# B&R Automation Studio project ACOPOStrak
Automation Studio 4.7.4.67 SP; technology packages: mapp 5.9.1, mappCockpit 5.9.0, mappMotion 5.9.2, mappView 5.9.1

## Configuration ACOPOStrak

### IoMap.iom - 5PC900_TS17_00/IoMap.iom
```iecst
VAR_CONFIG
	::gMain.status.safety.moduleOK AT %IX."epl_icn".ModuleOk;
	::gMain.status.safety.resetNeeded AT %IX."epl_icn".resetNeeded;
	::gMain.cmd.safety.reset AT %QX."epl_icn".resetCommand;
	::gMain.status.safety.started AT %IX."epl_icn".safetyStarted;
	::gMain.status.safety.ready AT %IX."epl_icn".safetyOK;
END_VAR
```

## Configuration Safety

CPU X20CP0484, AutomationRuntime C4.72, Build 4.1.2, Safety 0.0, Vc V4.72.0

### Task classes (Cpu.sw)
```
Cyclic#2 (cycle 20000 us, tolerance 20000 us):
  Safety <- Modules.Safety.Safety.prg
Binaries: arsvcreg, udbdef, TCData, arflatprv, arcoal, mvLoader, FWRules, mCoWebSc, ashwd, ashwac, User, sysconf, asfw, arconfig, Role, iomap, Config
Libraries: DataObj, AsXml, standard, runtime, FileIO, astime, mpbase, SfDomVis, asiodiag, asieccon, aruser, brsystem, SfDomDrv, sys_lib, MpSfDomMgr, asusb, astcp
```

### Hardware
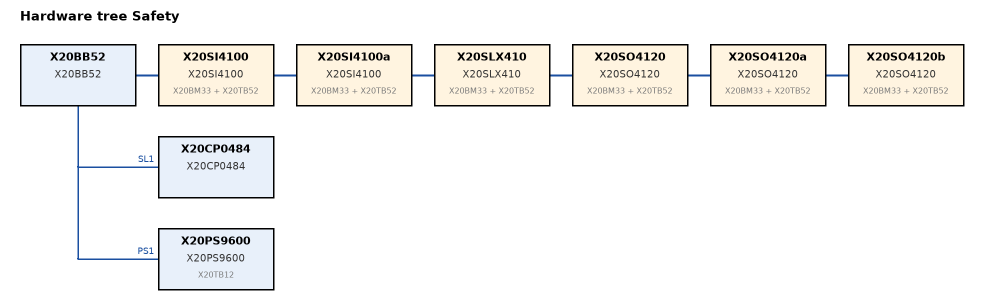
```
X20BB52 : X20BB52 v1.1.0.0
X20BM33 : X20BM33 v1.0.0.6  [X2X1 -> X20BB52.IF6]
X20BM33a : X20BM33 v1.0.0.6  [X2X1 -> X20BM33.X2X2]
X20BM33b : X20BM33 v1.0.0.6  [X2X1 -> X20BM33a.X2X2]
X20BM33c : X20BM33 v1.0.0.6  [X2X1 -> X20BM33b.X2X2]
X20BM33d : X20BM33 v1.0.0.6  [X2X1 -> X20BM33c.X2X2]
X20BM33e : X20BM33 v1.0.0.6  [X2X1 -> X20BM33d.X2X2]
X20CP0484 : X20CP0484 v1.2.1.0  [SL -> X20BB52.SL1]
  Connector IF2:
    ActivateDevice = 1
    Mode = Manual
    InternetAddress = 192.168.1.200
    SubnetMask = 255.255.255.0
  Connector IF3:
    CycleTime = 2400
    Mode = CN
    NodeID = 200
    EplNatSubnet = 192.168.103.0
    Channel1
    ChannelID1 = safetyStarted
    ChannelDirection1 = OUT
    Channel2
    ChannelID2 = safetyOK
    ChannelDirection2 = OUT
    Channel3
    ChannelID3 = resetNeeded
    ChannelDirection3 = OUT
    Channel4
    ChannelID4 = resetCommand
  ConfigurationID = ACOPOStrak_Safety
  TimerDeviceType = SWIOTIMER
  Cyclic1Duration = 2400
  Cyclic1Tolerance = 0
  Cyclic2Duration = 20000
  Cyclic2Tolerance = 20000
  Cyclic3Duration = 50000
  Cyclic3Tolerance = 50000
  Cyclic4Duration = 100000
  Cyclic4Tolerance = 100000
  Cyclic5Duration = 200000
  Cyclic5Tolerance = 200000
  Cyclic6Duration = 500000
  Cyclic6Tolerance = 500000
  Cyclic7Duration = 1000000
  Cyclic7Tolerance = 1000000
  Cyclic8Duration = 10000
  Cyclic8Tolerance = 30000000
X20PS9600 : X20PS9600 v1.0.1.0  [PS -> X20BB52.PS1; SS1 -> X20TB12.SS]
X20SI4100 : X20SI4100 v1.10.9.1  [SS1 -> X20TB52.SS; SL -> X20BM33.SL1]
  Supervision = off
X20SI4100a : X20SI4100 v1.10.9.1  [SS1 -> X20TB52a.SS; SL -> X20BM33a.SL1]
  Supervision = off
  SafeModuleID = 3
X20SLX410 : X20SLX410 v1.10.10.4  [SS1 -> X20TB52b.SS; SL -> X20BM33b.SL1]
  Supervision = off
X20SO4120 : X20SO4120 v1.10.9.1  [SS1 -> X20TB52c.SS; SL -> X20BM33c.SL1]
  Supervision = off
  SafeModuleID = 4
  DigitalOutput01 = viaSafeLOGIC
  DigitalOutput02 = viaSafeLOGIC
  DigitalOutput03 = viaSafeLOGIC
  DigitalOutput04 = viaSafeLOGIC
X20SO4120a : X20SO4120 v1.10.9.1  [SS1 -> X20TB52d.SS; SL -> X20BM33d.SL1]
  Supervision = off
  SafeModuleID = 5
  DigitalOutput01 = viaSafeLOGIC
  DigitalOutput02 = viaSafeLOGIC
  DigitalOutput03 = viaSafeLOGIC
  DigitalOutput04 = viaSafeLOGIC
X20SO4120b : X20SO4120 v1.10.9.1  [SS1 -> X20TB52e.SS; SL -> X20BM33e.SL1]
  Supervision = off
  SafeModuleID = 6
  DigitalOutput01 = viaSafeLOGIC
  DigitalOutput02 = viaSafeLOGIC
  DigitalOutput03 = viaSafeLOGIC
  DigitalOutput04 = viaSafeLOGIC
X20TB12 : X20TB12 v1.0.0.0
X20TB52 : X20TB52 v1.0.0.1
X20TB52a : X20TB52 v1.0.0.1
X20TB52b : X20TB52 v1.0.0.1
X20TB52c : X20TB52 v1.0.0.1
X20TB52d : X20TB52 v1.0.0.1
X20TB52e : X20TB52 v1.0.0.1
```

### IoMap.iom - X20CP0484/IoMap.iom
```iecst
VAR_CONFIG
	::Safety:this.cmd.reset AT %QX."X20SLX410".BOOL10001;
	::Safety:this.status.safetyStarted AT %IX."X20SLX410".BOOL00001;
	::Safety:this.status.safetyOk AT %IX."X20SLX410".BOOL00002;
	::Safety:this.status.resetNeeded AT %IX."X20SLX410".BOOL00003;
	::Safety:this.status.safetyStarted AT %QX."X20CP0484".IF3.safetyStarted;
	::Safety:this.status.safetyOk AT %QX."X20CP0484".IF3.safetyOK;
	::Safety:this.status.resetNeeded AT %QX."X20CP0484".IF3.resetNeeded;
	::Safety:this.cmd.reset AT %IX."X20CP0484".IF3.resetCommand;
END_VAR
```

- Safety project (password-protected, skipped)

## Configuration Simulation

CPU 5PC900.TS17-00, AutomationRuntime C4.72, Build 4.1.2, Safety 0.0, Vc V4.53.0

### Task classes (Cpu.sw)
```
Cyclic#1:
  Main <- Modules.Main.Main.prg
  Track1Sect <- Modules.Sectors.Track1Sector.Track1Sector.prg  // Task for handling Track 1 sectors
  Track2Sect <- Modules.Sectors.Track2Sector.Track2Sector.prg
  Track3Sect <- Modules.Sectors.Track3Sector.Track3Sector.prg  // Task for handling Track 3 sectors
  Track4Sect <- Modules.Sectors.Track4Sector.Track4Sector.prg  // Task for handling Track 4 sectors
  Track5Sect <- Modules.Sectors.Track5Sector.Track5Sector.prg
  Track6Sect <- Modules.Sectors.Track6Sector.Track6Sector.prg
Cyclic#8:
  Alarm <- Services.Alarm.Alarm.prg
  Simulation <- Simulation.Simulation.prg
DataObjects: McAcpSys
Binaries: TCData, udbdef, mvLoader, mCoWebSc, McAcpSim, arsvcreg, McAcpDrv, McProfGen, arflatprv, arcoal, Config_5, Config_4, AlarmCore, AlarmHist, Settings, ashwac, arconfig, asfw, TraceConfi, User, ashwd, iomap, Role, sysconf, Config_1, Config_3, Config_2
Libraries: McAxis, McBase, McAcpTrak, brdkMU, brsystem, AsSem, sys_lib, runtime, brdkSTR, operator, astime, AsIecCon, CoTrace, AsZip, FileIO, MpAlarmX, MpBase, MpAxis, McAcpAx, AsBrStr, AsIODiag, powerlnk, dataobj, MpSfDomMgr, SfDomDrv, SfDomVis, aruser, asusb, standard, astcp
```

### Hardware
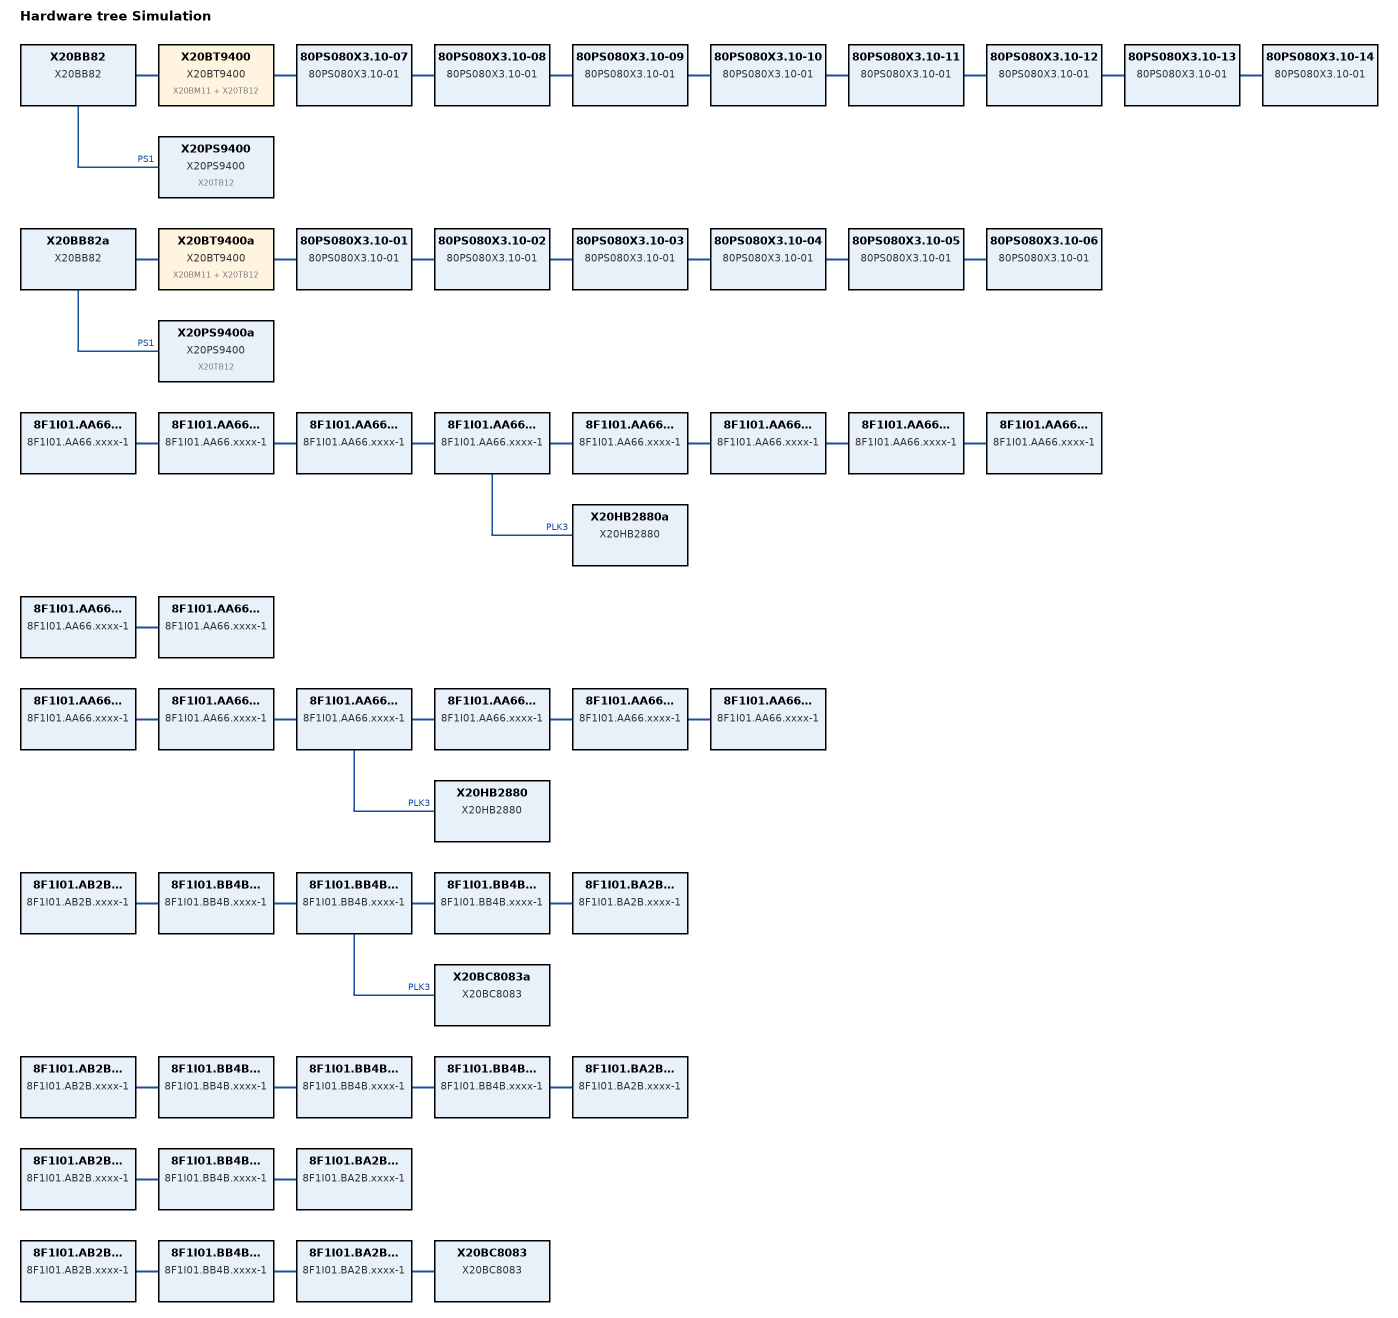
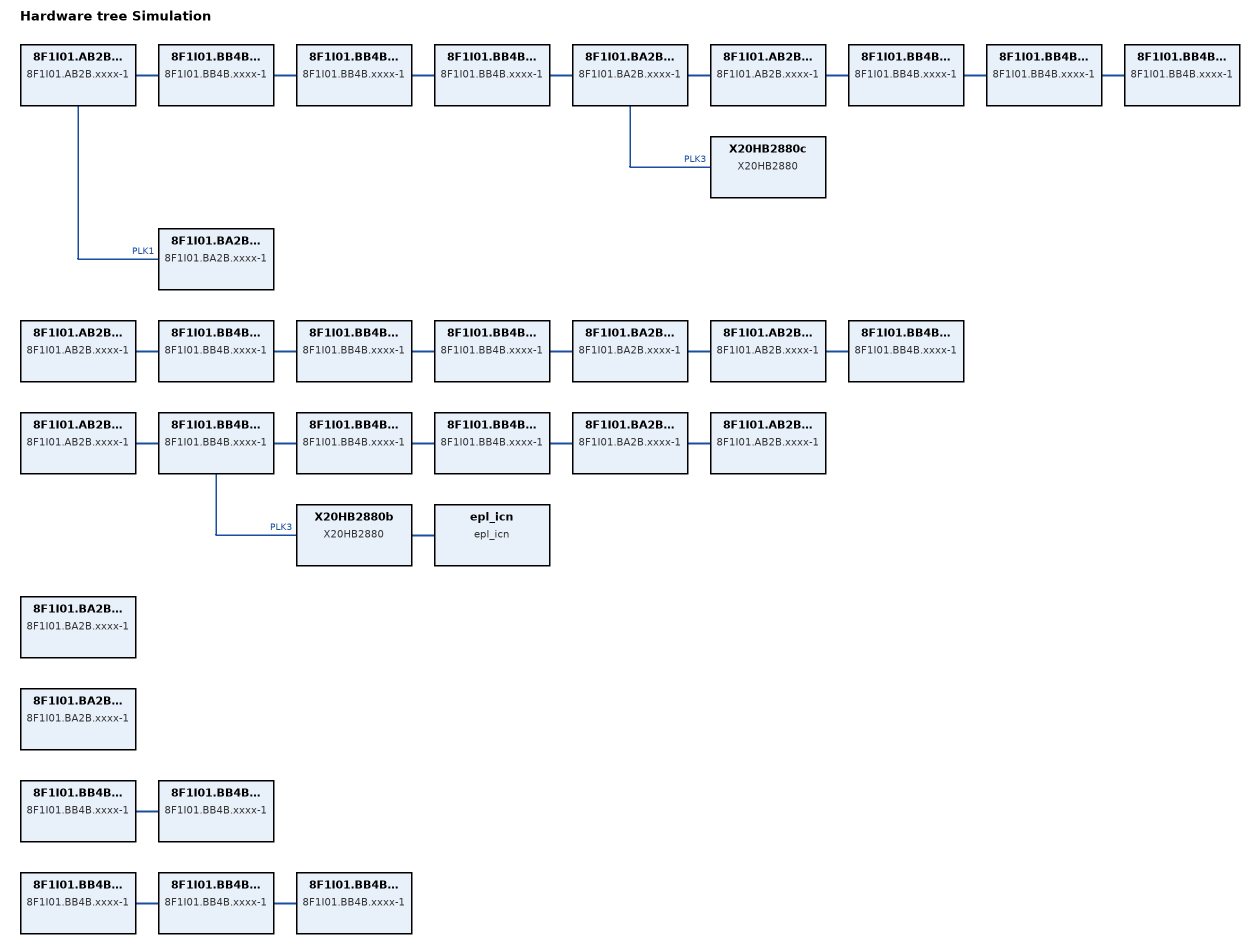
```
80PS080X3.10-01 : 80PS080X3.10-01 v1.3.0.0  [X2X1 -> X20BT9400a.X2X1 [Cable Type=X2XCable, Length=3, Version=1.0.0.2]]
  Supervision = off
  ParallelMode01 = on
  VoltageSet01 = 60
  ChopperEnable01 = on
80PS080X3.10-02 : 80PS080X3.10-01 v1.3.0.0  [X2X1 -> 80PS080X3.10-01.X2X2 [Cable Type=X2XCable, Length=1, Version=1.0.0.2]]
  Supervision = off
  ParallelMode01 = on
  VoltageSet01 = 60
  ChopperEnable01 = on
80PS080X3.10-03 : 80PS080X3.10-01 v1.3.0.0  [X2X1 -> 80PS080X3.10-02.X2X2 [Cable Type=X2XCable, Length=5, Version=1.0.0.2]]
  Supervision = off
  VoltageSet01 = 58
  ChopperEnable01 = on
80PS080X3.10-04 : 80PS080X3.10-01 v1.3.0.0  [X2X1 -> 80PS080X3.10-03.X2X2 [Cable Type=X2XCable, Length=1, Version=1.0.0.2]]
  Supervision = off
  VoltageSet01 = 58
  ChopperEnable01 = on
80PS080X3.10-05 : 80PS080X3.10-01 v1.3.0.0  [X2X1 -> 80PS080X3.10-04.X2X2 [Cable Type=X2XCable, Length=5, Version=1.0.0.2]]
  Supervision = off
  VoltageSet01 = 58
  ChopperEnable01 = on
80PS080X3.10-06 : 80PS080X3.10-01 v1.3.0.0  [X2X1 -> 80PS080X3.10-05.X2X2 [Cable Type=X2XCable, Length=1, Version=1.0.0.2]]
  Supervision = off
  VoltageSet01 = 58
  ChopperEnable01 = on
80PS080X3.10-07 : 80PS080X3.10-01 v1.3.0.0  [X2X1 -> X20BT9400.X2X1 [Cable Type=X2XCable, Length=5, Version=1.0.0.2]]
  Supervision = off
  VoltageSet01 = 58
  ChopperEnable01 = on
80PS080X3.10-08 : 80PS080X3.10-01 v1.3.0.0  [X2X1 -> 80PS080X3.10-07.X2X2 [Cable Type=X2XCable, Length=1, Version=1.0.0.2]]
  Supervision = off
  VoltageSet01 = 58
  ChopperEnable01 = on
80PS080X3.10-09 : 80PS080X3.10-01 v1.3.0.0  [X2X1 -> 80PS080X3.10-08.X2X2 [Cable Type=X2XCable, Length=1, Version=1.0.0.2]]
  Supervision = off
  VoltageSet01 = 58
  ChopperEnable01 = on
80PS080X3.10-10 : 80PS080X3.10-01 v1.3.0.0  [X2X1 -> 80PS080X3.10-09.X2X2 [Cable Type=X2XCable, Length=1, Version=1.0.0.2]]
  Supervision = off
  VoltageSet01 = 58
  ChopperEnable01 = on
80PS080X3.10-11 : 80PS080X3.10-01 v1.3.0.0  [X2X1 -> 80PS080X3.10-10.X2X2 [Cable Type=X2XCable, Length=3, Version=1.0.0.2]]
  Supervision = off
  VoltageSet01 = 58
  ChopperEnable01 = on
80PS080X3.10-12 : 80PS080X3.10-01 v1.3.0.0  [X2X1 -> 80PS080X3.10-11.X2X2 [Cable Type=X2XCable, Length=1, Version=1.0.0.2]]
  Supervision = off
  VoltageSet01 = 58
  ChopperEnable01 = on
80PS080X3.10-13 : 80PS080X3.10-01 v1.3.0.0  [X2X1 -> 80PS080X3.10-12.X2X2 [Cable Type=X2XCable, Length=1, Version=1.0.0.2]]
  Supervision = off
  VoltageSet01 = 58
  ChopperEnable01 = on
80PS080X3.10-14 : 80PS080X3.10-01 v1.3.0.0  [X2X1 -> 80PS080X3.10-13.X2X2 [Cable Type=X2XCable, Length=1, Version=1.0.0.2]]
  Supervision = off
  VoltageSet01 = 58
  ChopperEnable01 = on
8F1I01.AA66.xxxx-16 : 8F1I01.AA66.xxxx-1 v1.0.0.1  [PLK2 -> 8F1I01.AA66.xxxx-17.PLK1 (NodeNumber=16) [Cable Type=PowerlinkCable, Length=10, Version=1.0.0.2]]
  DriveConfiguration:
    McTypeID = LLMConfig
  DriveConfiguration/Segment:
    Shape = STRAIGHT660
    SegmentReference = SEG_1_16
    StopReaction = UseAssemblySetting
    SpeedFilter = UseAssemblySetting
8F1I01.AA66.xxxx-17 : 8F1I01.AA66.xxxx-1 v1.0.0.1  [PLK1 -> 8F1I01.AA66.xxxx-16.PLK2 (NodeNumber=17) [Cable Type=PowerlinkCable, Length=10, Version=1.0.0.2]; PLK2 -> 8F1I01.AA66.xxxx-18.PLK1 (NodeNumber=17) [Cable Type=PowerlinkCable, Length=10, Version=1.0.0.2]]
  DriveConfiguration:
    McTypeID = LLMConfig
  DriveConfiguration/Segment:
    Shape = STRAIGHT660
    SegmentReference = SEG_1_17
    StopReaction = UseAssemblySetting
    SpeedFilter = UseAssemblySetting
8F1I01.AA66.xxxx-18 : 8F1I01.AA66.xxxx-1 v1.0.0.1  [PLK1 -> 8F1I01.AA66.xxxx-17.PLK2 (NodeNumber=18) [Cable Type=PowerlinkCable, Length=10, Version=1.0.0.2]; PLK2 -> 8F1I01.AA66.xxxx-19.PLK1 (NodeNumber=18) [Cable Type=PowerlinkCable, Length=10, Version=1.0.0.2]]
  DriveConfiguration:
    McTypeID = LLMConfig
  DriveConfiguration/Segment:
    Shape = STRAIGHT660
    SegmentReference = SEG_1_18
    StopReaction = UseAssemblySetting
    SpeedFilter = UseAssemblySetting
8F1I01.AA66.xxxx-19 : 8F1I01.AA66.xxxx-1 v1.0.0.1  [PLK1 -> 8F1I01.AA66.xxxx-18.PLK2 (NodeNumber=19) [Cable Type=PowerlinkCable, Length=10, Version=1.0.0.2]; PLK2 -> 8F1I01.AA66.xxxx-20.PLK1 (NodeNumber=19) [Cable Type=PowerlinkCable, Length=10, Version=1.0.0.2]; PLK3 -> X20HB2880a.ETH1 (NodeNumber=19) [Cable Type=PowerlinkCable, Length=10, Version=1.0.0.2]]
  DriveConfiguration:
    McTypeID = LLMConfig
  DriveConfiguration/Segment:
    Shape = STRAIGHT660
    SegmentReference = SEG_1_19
    StopReaction = UseAssemblySetting
    SpeedFilter = UseAssemblySetting
8F1I01.AA66.xxxx-20 : 8F1I01.AA66.xxxx-1 v1.0.0.1  [PLK1 -> 8F1I01.AA66.xxxx-19.PLK2 (NodeNumber=20) [Cable Type=PowerlinkCable, Length=10, Version=1.0.0.2]; PLK2 -> 8F1I01.AA66.xxxx-21.PLK1 (NodeNumber=20) [Cable Type=PowerlinkCable, Length=10, Version=1.0.0.2]]
  DriveConfiguration:
    McTypeID = LLMConfig
  DriveConfiguration/Segment:
    Shape = STRAIGHT660
    SegmentReference = SEG_1_20
    StopReaction = UseAssemblySetting
    SpeedFilter = UseAssemblySetting
8F1I01.AA66.xxxx-21 : 8F1I01.AA66.xxxx-1 v1.0.0.1  [PLK1 -> 8F1I01.AA66.xxxx-20.PLK2 (NodeNumber=21) [Cable Type=PowerlinkCable, Length=10, Version=1.0.0.2]; PLK2 -> 8F1I01.AA66.xxxx-22.PLK1 (NodeNumber=21) [Cable Type=PowerlinkCable, Length=10, Version=1.0.0.2]]
  DriveConfiguration:
    McTypeID = LLMConfig
  DriveConfiguration/Segment:
    Shape = STRAIGHT660
    SegmentReference = SEG_1_21
    StopReaction = UseAssemblySetting
    SpeedFilter = UseAssemblySetting
8F1I01.AA66.xxxx-22 : 8F1I01.AA66.xxxx-1 v1.0.0.1  [PLK1 -> 8F1I01.AA66.xxxx-21.PLK2 (NodeNumber=22) [Cable Type=PowerlinkCable, Length=10, Version=1.0.0.2]; PLK2 -> 8F1I01.AA66.xxxx-23.PLK1 (NodeNumber=22) [Cable Type=PowerlinkCable, Length=10, Version=1.0.0.2]]
  DriveConfiguration:
    McTypeID = LLMConfig
  DriveConfiguration/Segment:
    Shape = STRAIGHT660
    SegmentReference = SEG_1_22
    StopReaction = UseAssemblySetting
    SpeedFilter = UseAssemblySetting
8F1I01.AA66.xxxx-23 : 8F1I01.AA66.xxxx-1 v1.0.0.1  [PLK1 -> 8F1I01.AA66.xxxx-22.PLK2 (NodeNumber=23) [Cable Type=PowerlinkCable, Length=10, Version=1.0.0.2]]
  DriveConfiguration:
    McTypeID = LLMConfig
  DriveConfiguration/Segment:
    Shape = STRAIGHT660
    SegmentReference = SEG_1_23
    StopReaction = UseAssemblySetting
    SpeedFilter = UseAssemblySetting
8F1I01.AA66.xxxx-29 : 8F1I01.AA66.xxxx-1 v1.0.0.1  [PLK1 -> 8F1I01.BA2B.xxxx-28.PLK2 (NodeNumber=29) [Cable Type=PowerlinkCable, Length=10, Version=1.0.0.2]; PLK2 -> 8F1I01.AA66.xxxx-30.PLK1 (NodeNumber=29) [Cable Type=PowerlinkCable, Length=10, Version=1.0.0.2]]
  DriveConfiguration:
    McTypeID = LLMConfig
  DriveConfiguration/Segment:
    Shape = STRAIGHT660
    SegmentReference = SEG_1_29
    StopReaction = UseAssemblySetting
    SpeedFilter = UseAssemblySetting
8F1I01.AA66.xxxx-30 : 8F1I01.AA66.xxxx-1 v1.0.0.1  [PLK1 -> 8F1I01.AA66.xxxx-29.PLK2 (NodeNumber=30) [Cable Type=PowerlinkCable, Length=10, Version=1.0.0.2]]
  DriveConfiguration:
    McTypeID = LLMConfig
  DriveConfiguration/Segment:
    Shape = STRAIGHT660
    SegmentReference = SEG_1_30
    StopReaction = UseAssemblySetting
    SpeedFilter = UseAssemblySetting
8F1I01.AA66.xxxx-31 : 8F1I01.AA66.xxxx-1 v1.0.0.1  [PLK2 -> 8F1I01.AA66.xxxx-32.PLK1 (NodeNumber=31) [Cable Type=PowerlinkCable, Length=10, Version=1.0.0.2]]
  DriveConfiguration:
    McTypeID = LLMConfig
  DriveConfiguration/Segment:
    Shape = STRAIGHT660
    SegmentReference = SEG_1_31
    StopReaction = UseAssemblySetting
    SpeedFilter = UseAssemblySetting
8F1I01.AA66.xxxx-32 : 8F1I01.AA66.xxxx-1 v1.0.0.1  [PLK1 -> 8F1I01.AA66.xxxx-31.PLK2 (NodeNumber=32) [Cable Type=PowerlinkCable, Length=10, Version=1.0.0.2]; PLK2 -> 8F1I01.AA66.xxxx-33.PLK1 (NodeNumber=32) [Cable Type=PowerlinkCable, Length=10, Version=1.0.0.2]]
  DriveConfiguration:
    McTypeID = LLMConfig
  DriveConfiguration/Segment:
    Shape = STRAIGHT660
    SegmentReference = SEG_1_32
    StopReaction = UseAssemblySetting
    SpeedFilter = UseAssemblySetting
8F1I01.AA66.xxxx-33 : 8F1I01.AA66.xxxx-1 v1.0.0.1  [PLK1 -> 8F1I01.AA66.xxxx-32.PLK2 (NodeNumber=33) [Cable Type=PowerlinkCable, Length=10, Version=1.0.0.2]; PLK2 -> 8F1I01.AA66.xxxx-34.PLK1 (NodeNumber=33) [Cable Type=PowerlinkCable, Length=10, Version=1.0.0.2]; PLK3 -> X20HB2880.ETH1 (NodeNumber=33) [Cable Type=PowerlinkCable, Length=10, Version=1.0.0.2]]
  DriveConfiguration:
    McTypeID = LLMConfig
  DriveConfiguration/Segment:
    Shape = STRAIGHT660
    SegmentReference = SEG_1_33
    StopReaction = UseAssemblySetting
    SpeedFilter = UseAssemblySetting
8F1I01.AA66.xxxx-34 : 8F1I01.AA66.xxxx-1 v1.0.0.1  [PLK1 -> 8F1I01.AA66.xxxx-33.PLK2 (NodeNumber=34) [Cable Type=PowerlinkCable, Length=10, Version=1.0.0.2]; PLK2 -> 8F1I01.AA66.xxxx-35.PLK1 (NodeNumber=34) [Cable Type=PowerlinkCable, Length=10, Version=1.0.0.2]]
  DriveConfiguration:
    McTypeID = LLMConfig
  DriveConfiguration/Segment:
    Shape = STRAIGHT660
    SegmentReference = SEG_1_34
    StopReaction = UseAssemblySetting
    SpeedFilter = UseAssemblySetting
8F1I01.AA66.xxxx-35 : 8F1I01.AA66.xxxx-1 v1.0.0.1  [PLK1 -> 8F1I01.AA66.xxxx-34.PLK2 (NodeNumber=35) [Cable Type=PowerlinkCable, Length=10, Version=1.0.0.2]; PLK2 -> 8F1I01.AA66.xxxx-36.PLK1 (NodeNumber=35) [Cable Type=PowerlinkCable, Length=10, Version=1.0.0.2]]
  DriveConfiguration:
    McTypeID = LLMConfig
  DriveConfiguration/Segment:
    Shape = STRAIGHT660
    SegmentReference = SEG_1_35
    StopReaction = UseAssemblySetting
    SpeedFilter = UseAssemblySetting
8F1I01.AA66.xxxx-36 : 8F1I01.AA66.xxxx-1 v1.0.0.1  [PLK1 -> 8F1I01.AA66.xxxx-35.PLK2 (NodeNumber=36) [Cable Type=PowerlinkCable, Length=10, Version=1.0.0.2]]
  DriveConfiguration:
    McTypeID = LLMConfig
  DriveConfiguration/Segment:
    Shape = STRAIGHT660
    SegmentReference = SEG_1_36
    StopReaction = UseAssemblySetting
    SpeedFilter = UseAssemblySetting
8F1I01.AB2B.xxxx-11 : 8F1I01.AB2B.xxxx-1 v1.0.0.1  [PLK2 -> 8F1I01.BB4B.xxxx-12.PLK1 (NodeNumber=11) [Cable Type=PowerlinkCable, Length=10, Version=1.0.0.2]]
  DriveConfiguration:
    McTypeID = LLMConfig
  DriveConfiguration/Segment:
    Shape = STRAIGHT105_TO_CIRCULAR
    SegmentReference = SEG_1_11
    StopReaction = UseAssemblySetting
    SpeedFilter = UseAssemblySetting
8F1I01.AB2B.xxxx-24 : 8F1I01.AB2B.xxxx-1 v1.0.0.1  [PLK2 -> 8F1I01.BB4B.xxxx-25.PLK1 (NodeNumber=24) [Cable Type=PowerlinkCable, Length=10, Version=1.0.0.2]]
  DriveConfiguration:
    McTypeID = LLMConfig
  DriveConfiguration/Segment:
    Shape = STRAIGHT105_TO_CIRCULAR
    SegmentReference = SEG_1_24
    StopReaction = UseAssemblySetting
    SpeedFilter = UseAssemblySetting
8F1I01.AB2B.xxxx-37 : 8F1I01.AB2B.xxxx-1 v1.0.0.1  [PLK2 -> 8F1I01.BB4B.xxxx-38.PLK1 (NodeNumber=37) [Cable Type=PowerlinkCable, Length=10, Version=1.0.0.2]; PLK3 -> X20HB2880.ETH2 (NodeNumber=37) [Cable Type=PowerlinkCable, Length=10, Version=1.0.0.2]]
  DriveConfiguration:
    McTypeID = LLMConfig
  DriveConfiguration/Segment:
    Shape = STRAIGHT105_TO_CIRCULAR
    SegmentReference = SEG_5_37
    StopReaction = UseAssemblySetting
    SpeedFilter = UseAssemblySetting
8F1I01.AB2B.xxxx-51 : 8F1I01.AB2B.xxxx-1 v1.0.0.1  [PLK2 -> 8F1I01.BB4B.xxxx-52.PLK1 (NodeNumber=51) [Cable Type=PowerlinkCable, Length=10, Version=1.0.0.2]]
  DriveConfiguration:
    McTypeID = LLMConfig
  DriveConfiguration/Segment:
    Shape = STRAIGHT105_TO_CIRCULAR
    SegmentReference = SEG_6_51
    StopReaction = UseAssemblySetting
    SpeedFilter = UseAssemblySetting
8F1I01.AB2B.xxxx-55 : 8F1I01.AB2B.xxxx-1 v1.0.0.1  [PLK1 -> 8F1I01.BA2B.xxxx-54.PLK2 (NodeNumber=55) [Cable Type=PowerlinkCable, Length=10, Version=1.0.0.2]; PLK2 -> 8F1I01.BB4B.xxxx-56.PLK1 (NodeNumber=55) [Cable Type=PowerlinkCable, Length=10, Version=1.0.0.2]]
  DriveConfiguration:
    McTypeID = LLMConfig
  DriveConfiguration/Segment:
    Shape = STRAIGHT105_TO_CIRCULAR
    SegmentReference = SEG_4_55
    StopReaction = UseAssemblySetting
    SpeedFilter = UseAssemblySetting
8F1I01.AB2B.xxxx-60 : 8F1I01.AB2B.xxxx-1 v1.0.0.1  [PLK1 -> 8F1I01.BA2B.xxxx-59.PLK2 (NodeNumber=60) [Cable Type=PowerlinkCable, Length=10, Version=1.0.0.2]; PLK2 -> 8F1I01.BB4B.xxxx-61.PLK1 (NodeNumber=60) [Cable Type=PowerlinkCable, Length=10, Version=1.0.0.2]]
  DriveConfiguration:
    McTypeID = LLMConfig
  DriveConfiguration/Segment:
    Shape = STRAIGHT105_TO_CIRCULAR
    SegmentReference = SEG_4_60
    StopReaction = UseAssemblySetting
    SpeedFilter = UseAssemblySetting
8F1I01.AB2B.xxxx-67 : 8F1I01.AB2B.xxxx-1 v1.0.0.1  [PLK1 -> 8F1I01.BA2B.xxxx-66.PLK2 (NodeNumber=67) [Cable Type=PowerlinkCable, Length=10, Version=1.0.0.2]; PLK2 -> 8F1I01.BB4B.xxxx-68.PLK1 (NodeNumber=67) [Cable Type=PowerlinkCable, Length=10, Version=1.0.0.2]]
  DriveConfiguration:
    McTypeID = LLMConfig
  DriveConfiguration/Segment:
    Shape = STRAIGHT105_TO_CIRCULAR
    SegmentReference = SEG_3_67
    StopReaction = UseAssemblySetting
    SpeedFilter = UseAssemblySetting
8F1I01.AB2B.xxxx-72 : 8F1I01.AB2B.xxxx-1 v1.0.0.1  [PLK1 -> 8F1I01.BA2B.xxxx-71.PLK2 (NodeNumber=72) [Cable Type=PowerlinkCable, Length=10, Version=1.0.0.2]; PLK2 -> 8F1I01.BB4B.xxxx-73.PLK1 (NodeNumber=72) [Cable Type=PowerlinkCable, Length=10, Version=1.0.0.2]]
  DriveConfiguration:
    McTypeID = LLMConfig
  DriveConfiguration/Segment:
    Shape = STRAIGHT105_TO_CIRCULAR
    SegmentReference = SEG_3_72
    StopReaction = UseAssemblySetting
    SpeedFilter = UseAssemblySetting
8F1I01.AB2B.xxxx-78 : 8F1I01.AB2B.xxxx-1 v1.0.0.1  [PLK1 -> 8F1I01.BA2B.xxxx-77.PLK2 (NodeNumber=78) [Cable Type=PowerlinkCable, Length=10, Version=1.0.0.2]; PLK2 -> 8F1I01.BB4B.xxxx-79.PLK1 (NodeNumber=78) [Cable Type=PowerlinkCable, Length=10, Version=1.0.0.2]]
  DriveConfiguration:
    McTypeID = LLMConfig
  DriveConfiguration/Segment:
    Shape = STRAIGHT105_TO_CIRCULAR
    SegmentReference = SEG_2_78
    StopReaction = UseAssemblySetting
    SpeedFilter = UseAssemblySetting
8F1I01.AB2B.xxxx-83 : 8F1I01.AB2B.xxxx-1 v1.0.0.1  [PLK1 -> 8F1I01.BA2B.xxxx-82.PLK2 (NodeNumber=83) [Cable Type=PowerlinkCable, Length=10, Version=1.0.0.2]]
  DriveConfiguration:
    McTypeID = LLMConfig
  DriveConfiguration/Segment:
    Shape = STRAIGHT105_TO_CIRCULAR
    SegmentReference = SEG_2_83
    StopReaction = UseAssemblySetting
    SpeedFilter = UseAssemblySetting
8F1I01.BA2B.xxxx-15 : 8F1I01.BA2B.xxxx-1 v1.0.0.1  [PLK1 -> 8F1I01.BB4B.xxxx-14.PLK2 (NodeNumber=15) [Cable Type=PowerlinkCable, Length=10, Version=1.0.0.2]]
  DriveConfiguration:
    McTypeID = LLMConfig
  DriveConfiguration/Segment:
    Shape = CIRCULAR_TO_STRAIGHT105
    SegmentReference = SEG_1_15
    StopReaction = UseAssemblySetting
    SpeedFilter = UseAssemblySetting
8F1I01.BA2B.xxxx-28 : 8F1I01.BA2B.xxxx-1 v1.0.0.1  [PLK1 -> 8F1I01.BB4B.xxxx-27.PLK2 (NodeNumber=28) [Cable Type=PowerlinkCable, Length=10, Version=1.0.0.2]; PLK2 -> 8F1I01.AA66.xxxx-29.PLK1 (NodeNumber=28) [Cable Type=PowerlinkCable, Length=10, Version=1.0.0.2]; PLK3 -> X20HB2880a.ETH2 (NodeNumber=28) [Cable Type=PowerlinkCable, Length=10, Version=1.0.0.2]]
  DriveConfiguration:
    McTypeID = LLMConfig
  DriveConfiguration/Segment:
    Shape = CIRCULAR_TO_STRAIGHT105
    SegmentReference = SEG_1_28
    StopReaction = UseAssemblySetting
    SpeedFilter = UseAssemblySetting
8F1I01.BA2B.xxxx-39 : 8F1I01.BA2B.xxxx-1 v1.0.0.1  [PLK1 -> 8F1I01.BB4B.xxxx-38.PLK2 (NodeNumber=39) [Cable Type=PowerlinkCable, Length=10, Version=1.0.0.2]]
  DriveConfiguration:
    McTypeID = LLMConfig
  DriveConfiguration/Segment:
    Shape = CIRCULAR_TO_STRAIGHT105
    SegmentReference = SEG_5_39
    StopReaction = UseAssemblySetting
    SpeedFilter = UseAssemblySetting
8F1I01.BA2B.xxxx-53 : 8F1I01.BA2B.xxxx-1 v1.0.0.1  [PLK1 -> 8F1I01.BB4B.xxxx-52.PLK2 (NodeNumber=53) [Cable Type=PowerlinkCable, Length=10, Version=1.0.0.2]; PLK3 -> X20BC8083.PLK2 (NodeNumber=53) [Cable Type=PowerlinkCable, Length=10, Version=1.0.0.2]]
  DriveConfiguration:
    McTypeID = LLMConfig
  DriveConfiguration/Segment:
    Shape = CIRCULAR_TO_STRAIGHT105
    SegmentReference = SEG_6_53
    StopReaction = UseAssemblySetting
    SpeedFilter = UseAssemblySetting
8F1I01.BA2B.xxxx-54 : 8F1I01.BA2B.xxxx-1 v1.0.0.1  [PLK2 -> 8F1I01.AB2B.xxxx-55.PLK1 (NodeNumber=54) [Cable Type=PowerlinkCable, Length=10, Version=1.0.0.2]]
  DriveConfiguration:
    McTypeID = LLMConfig
  DriveConfiguration/Segment:
    Shape = CIRCULAR_TO_STRAIGHT105
    SegmentReference = SEG_4_54
    StopReaction = UseAssemblySetting
    SpeedFilter = UseAssemblySetting
8F1I01.BA2B.xxxx-59 : 8F1I01.BA2B.xxxx-1 v1.0.0.1  [PLK1 -> 8F1I01.BB4B.xxxx-58.PLK2 (NodeNumber=59) [Cable Type=PowerlinkCable, Length=10, Version=1.0.0.2]; PLK2 -> 8F1I01.AB2B.xxxx-60.PLK1 (NodeNumber=59) [Cable Type=PowerlinkCable, Length=10, Version=1.0.0.2]; PLK3 -> X20HB2880c.ETH1 (NodeNumber=59) [Cable Type=PowerlinkCable, Length=10, Version=1.0.0.2]]
  DriveConfiguration:
    McTypeID = LLMConfig
  DriveConfiguration/Segment:
    Shape = CIRCULAR_TO_STRAIGHT105
    SegmentReference = SEG_4_59
    StopReaction = UseAssemblySetting
    SpeedFilter = UseAssemblySetting
8F1I01.BA2B.xxxx-66 : 8F1I01.BA2B.xxxx-1 v1.0.0.1  [PLK1 -> 8F1I01.BB4B.xxxx-65.PLK2 (NodeNumber=66) [Cable Type=PowerlinkCable, Length=10, Version=1.0.0.2]; PLK2 -> 8F1I01.AB2B.xxxx-67.PLK1 (NodeNumber=66) [Cable Type=PowerlinkCable, Length=10, Version=1.0.0.2]]
  DriveConfiguration:
    McTypeID = LLMConfig
  DriveConfiguration/Segment:
    Shape = CIRCULAR_TO_STRAIGHT105
    SegmentReference = SEG_3_66
    StopReaction = UseAssemblySetting
    SpeedFilter = UseAssemblySetting
8F1I01.BA2B.xxxx-71 : 8F1I01.BA2B.xxxx-1 v1.0.0.1  [PLK1 -> 8F1I01.BB4B.xxxx-70.PLK2 (NodeNumber=71) [Cable Type=PowerlinkCable, Length=10, Version=1.0.0.2]; PLK2 -> 8F1I01.AB2B.xxxx-72.PLK1 (NodeNumber=71) [Cable Type=PowerlinkCable, Length=10, Version=1.0.0.2]]
  DriveConfiguration:
    McTypeID = LLMConfig
  DriveConfiguration/Segment:
    Shape = CIRCULAR_TO_STRAIGHT105
    SegmentReference = SEG_3_71
    StopReaction = UseAssemblySetting
    SpeedFilter = UseAssemblySetting
8F1I01.BA2B.xxxx-77 : 8F1I01.BA2B.xxxx-1 v1.0.0.1  [PLK1 -> 8F1I01.BB4B.xxxx-76.PLK2 (NodeNumber=77) [Cable Type=PowerlinkCable, Length=10, Version=1.0.0.2]; PLK2 -> 8F1I01.AB2B.xxxx-78.PLK1 (NodeNumber=77) [Cable Type=PowerlinkCable, Length=10, Version=1.0.0.2]]
  DriveConfiguration:
    McTypeID = LLMConfig
  DriveConfiguration/Segment:
    Shape = CIRCULAR_TO_STRAIGHT105
    SegmentReference = SEG_2_77
    StopReaction = UseAssemblySetting
    SpeedFilter = UseAssemblySetting
8F1I01.BA2B.xxxx-82 : 8F1I01.BA2B.xxxx-1 v1.0.0.1  [PLK1 -> 8F1I01.BB4B.xxxx-81.PLK2 (NodeNumber=82) [Cable Type=PowerlinkCable, Length=10, Version=1.0.0.2]; PLK2 -> 8F1I01.AB2B.xxxx-83.PLK1 (NodeNumber=82) [Cable Type=PowerlinkCable, Length=10, Version=1.0.0.2]]
  DriveConfiguration:
    McTypeID = LLMConfig
  DriveConfiguration/Segment:
    Shape = CIRCULAR_TO_STRAIGHT105
    SegmentReference = SEG_2_82
    StopReaction = UseAssemblySetting
    SpeedFilter = UseAssemblySetting
8F1I01.BB4B.xxxx-12 : 8F1I01.BB4B.xxxx-1 v1.0.0.1  [PLK1 -> 8F1I01.AB2B.xxxx-11.PLK2 (NodeNumber=12) [Cable Type=PowerlinkCable, Length=10, Version=1.0.0.2]; PLK2 -> 8F1I01.BB4B.xxxx-13.PLK1 (NodeNumber=12) [Cable Type=PowerlinkCable, Length=10, Version=1.0.0.2]]
  DriveConfiguration:
    McTypeID = LLMConfig
  DriveConfiguration/Segment:
    Shape = CIRCULAR
    SegmentReference = SEG_1_12
    StopReaction = UseAssemblySetting
    SpeedFilter = UseAssemblySetting
8F1I01.BB4B.xxxx-13 : 8F1I01.BB4B.xxxx-1 v1.0.0.1  [PLK1 -> 8F1I01.BB4B.xxxx-12.PLK2 (NodeNumber=13) [Cable Type=PowerlinkCable, Length=10, Version=1.0.0.2]; PLK2 -> 8F1I01.BB4B.xxxx-14.PLK1 (NodeNumber=13) [Cable Type=PowerlinkCable, Length=10, Version=1.0.0.2]; PLK3 -> X20BC8083a.PLK2 (NodeNumber=13) [Cable Type=PowerlinkCable, Length=10, Version=1.0.0.2]]
  DriveConfiguration:
    McTypeID = LLMConfig
  DriveConfiguration/Segment:
    Shape = CIRCULAR
    SegmentReference = SEG_1_13
    StopReaction = UseAssemblySetting
    SpeedFilter = UseAssemblySetting
8F1I01.BB4B.xxxx-14 : 8F1I01.BB4B.xxxx-1 v1.0.0.1  [PLK1 -> 8F1I01.BB4B.xxxx-13.PLK2 (NodeNumber=14) [Cable Type=PowerlinkCable, Length=10, Version=1.0.0.2]; PLK2 -> 8F1I01.BA2B.xxxx-15.PLK1 (NodeNumber=14) [Cable Type=PowerlinkCable, Length=10, Version=1.0.0.2]]
  DriveConfiguration:
    McTypeID = LLMConfig
  DriveConfiguration/Segment:
    Shape = CIRCULAR
    SegmentReference = SEG_1_14
    StopReaction = UseAssemblySetting
    SpeedFilter = UseAssemblySetting
8F1I01.BB4B.xxxx-25 : 8F1I01.BB4B.xxxx-1 v1.0.0.1  [PLK1 -> 8F1I01.AB2B.xxxx-24.PLK2 (NodeNumber=25) [Cable Type=PowerlinkCable, Length=10, Version=1.0.0.2]; PLK2 -> 8F1I01.BB4B.xxxx-26.PLK1 (NodeNumber=25) [Cable Type=PowerlinkCable, Length=10, Version=1.0.0.2]]
  DriveConfiguration:
    McTypeID = LLMConfig
  DriveConfiguration/Segment:
    Shape = CIRCULAR
    SegmentReference = SEG_1_25
    StopReaction = UseAssemblySetting
    SpeedFilter = UseAssemblySetting
8F1I01.BB4B.xxxx-26 : 8F1I01.BB4B.xxxx-1 v1.0.0.1  [PLK1 -> 8F1I01.BB4B.xxxx-25.PLK2 (NodeNumber=26) [Cable Type=PowerlinkCable, Length=10, Version=1.0.0.2]; PLK2 -> 8F1I01.BB4B.xxxx-27.PLK1 (NodeNumber=26) [Cable Type=PowerlinkCable, Length=10, Version=1.0.0.2]]
  DriveConfiguration:
    McTypeID = LLMConfig
  DriveConfiguration/Segment:
    Shape = CIRCULAR
    SegmentReference = SEG_1_26
    StopReaction = UseAssemblySetting
    SpeedFilter = UseAssemblySetting
8F1I01.BB4B.xxxx-27 : 8F1I01.BB4B.xxxx-1 v1.0.0.1  [PLK1 -> 8F1I01.BB4B.xxxx-26.PLK2 (NodeNumber=27) [Cable Type=PowerlinkCable, Length=10, Version=1.0.0.2]; PLK2 -> 8F1I01.BA2B.xxxx-28.PLK1 (NodeNumber=27) [Cable Type=PowerlinkCable, Length=10, Version=1.0.0.2]]
  DriveConfiguration:
    McTypeID = LLMConfig
  DriveConfiguration/Segment:
    Shape = CIRCULAR
    SegmentReference = SEG_1_27
    StopReaction = UseAssemblySetting
    SpeedFilter = UseAssemblySetting
8F1I01.BB4B.xxxx-38 : 8F1I01.BB4B.xxxx-1 v1.0.0.1  [PLK1 -> 8F1I01.AB2B.xxxx-37.PLK2 (NodeNumber=38) [Cable Type=PowerlinkCable, Length=10, Version=1.0.0.2]; PLK2 -> 8F1I01.BA2B.xxxx-39.PLK1 (NodeNumber=38) [Cable Type=PowerlinkCable, Length=10, Version=1.0.0.2]]
  DriveConfiguration:
    McTypeID = LLMConfig
  DriveConfiguration/Segment:
    Shape = CIRCULAR
    SegmentReference = SEG_5_38
    StopReaction = UseAssemblySetting
    SpeedFilter = UseAssemblySetting
8F1I01.BB4B.xxxx-52 : 8F1I01.BB4B.xxxx-1 v1.0.0.1  [PLK1 -> 8F1I01.AB2B.xxxx-51.PLK2 (NodeNumber=52) [Cable Type=PowerlinkCable, Length=10, Version=1.0.0.2]; PLK2 -> 8F1I01.BA2B.xxxx-53.PLK1 (NodeNumber=52) [Cable Type=PowerlinkCable, Length=10, Version=1.0.0.2]]
  DriveConfiguration:
    McTypeID = LLMConfig
  DriveConfiguration/Segment:
    Shape = CIRCULAR
    SegmentReference = SEG_6_52
    StopReaction = UseAssemblySetting
    SpeedFilter = UseAssemblySetting
8F1I01.BB4B.xxxx-56 : 8F1I01.BB4B.xxxx-1 v1.0.0.1  [PLK1 -> 8F1I01.AB2B.xxxx-55.PLK2 (NodeNumber=56) [Cable Type=PowerlinkCable, Length=10, Version=1.0.0.2]; PLK2 -> 8F1I01.BB4B.xxxx-57.PLK1 (NodeNumber=56) [Cable Type=PowerlinkCable, Length=10, Version=1.0.0.2]]
  DriveConfiguration:
    McTypeID = LLMConfig
  DriveConfiguration/Segment:
    Shape = CIRCULAR
    SegmentReference = SEG_4_56
    StopReaction = UseAssemblySetting
    SpeedFilter = UseAssemblySetting
8F1I01.BB4B.xxxx-57 : 8F1I01.BB4B.xxxx-1 v1.0.0.1  [PLK1 -> 8F1I01.BB4B.xxxx-56.PLK2 (NodeNumber=57) [Cable Type=PowerlinkCable, Length=10, Version=1.0.0.2]; PLK2 -> 8F1I01.BB4B.xxxx-58.PLK1 (NodeNumber=57) [Cable Type=PowerlinkCable, Length=10, Version=1.0.0.2]]
  DriveConfiguration:
    McTypeID = LLMConfig
  DriveConfiguration/Segment:
    Shape = CIRCULAR
    SegmentReference = SEG_4_57
    StopReaction = UseAssemblySetting
    SpeedFilter = UseAssemblySetting
8F1I01.BB4B.xxxx-58 : 8F1I01.BB4B.xxxx-1 v1.0.0.1  [PLK1 -> 8F1I01.BB4B.xxxx-57.PLK2 (NodeNumber=58) [Cable Type=PowerlinkCable, Length=10, Version=1.0.0.2]; PLK2 -> 8F1I01.BA2B.xxxx-59.PLK1 (NodeNumber=58) [Cable Type=PowerlinkCable, Length=10, Version=1.0.0.2]]
  DriveConfiguration:
    McTypeID = LLMConfig
  DriveConfiguration/Segment:
    Shape = CIRCULAR
    SegmentReference = SEG_4_58
    StopReaction = UseAssemblySetting
    SpeedFilter = UseAssemblySetting
8F1I01.BB4B.xxxx-61 : 8F1I01.BB4B.xxxx-1 v1.0.0.1  [PLK1 -> 8F1I01.AB2B.xxxx-60.PLK2 (NodeNumber=61) [Cable Type=PowerlinkCable, Length=10, Version=1.0.0.2]; PLK2 -> 8F1I01.BB4B.xxxx-62.PLK1 (NodeNumber=61) [Cable Type=PowerlinkCable, Length=10, Version=1.0.0.2]]
  DriveConfiguration:
    McTypeID = LLMConfig
  DriveConfiguration/Segment:
    Shape = CIRCULAR
    SegmentReference = SEG_4_61
    StopReaction = UseAssemblySetting
    SpeedFilter = UseAssemblySetting
8F1I01.BB4B.xxxx-62 : 8F1I01.BB4B.xxxx-1 v1.0.0.1  [PLK1 -> 8F1I01.BB4B.xxxx-61.PLK2 (NodeNumber=62) [Cable Type=PowerlinkCable, Length=10, Version=1.0.0.2]; PLK2 -> 8F1I01.BB4B.xxxx-63.PLK1 (NodeNumber=62) [Cable Type=PowerlinkCable, Length=10, Version=1.0.0.2]]
  DriveConfiguration:
    McTypeID = LLMConfig
  DriveConfiguration/Segment:
    Shape = CIRCULAR
    SegmentReference = SEG_4_62
    StopReaction = UseAssemblySetting
    SpeedFilter = UseAssemblySetting
8F1I01.BB4B.xxxx-63 : 8F1I01.BB4B.xxxx-1 v1.0.0.1  [PLK1 -> 8F1I01.BB4B.xxxx-62.PLK2 (NodeNumber=63) [Cable Type=PowerlinkCable, Length=10, Version=1.0.0.2]]
  DriveConfiguration:
    McTypeID = LLMConfig
  DriveConfiguration/Segment:
    Shape = CIRCULAR
    SegmentReference = SEG_4_63
    StopReaction = UseAssemblySetting
    SpeedFilter = UseAssemblySetting
8F1I01.BB4B.xxxx-64 : 8F1I01.BB4B.xxxx-1 v1.0.0.1  [PLK2 -> 8F1I01.BB4B.xxxx-65.PLK1 (NodeNumber=64) [Cable Type=PowerlinkCable, Length=10, Version=1.0.0.2]]
  DriveConfiguration:
    McTypeID = LLMConfig
  DriveConfiguration/Segment:
    Shape = CIRCULAR
    SegmentReference = SEG_3_64
    StopReaction = UseAssemblySetting
    SpeedFilter = UseAssemblySetting
8F1I01.BB4B.xxxx-65 : 8F1I01.BB4B.xxxx-1 v1.0.0.1  [PLK1 -> 8F1I01.BB4B.xxxx-64.PLK2 (NodeNumber=65) [Cable Type=PowerlinkCable, Length=10, Version=1.0.0.2]; PLK2 -> 8F1I01.BA2B.xxxx-66.PLK1 (NodeNumber=65) [Cable Type=PowerlinkCable, Length=10, Version=1.0.0.2]]
  DriveConfiguration:
    McTypeID = LLMConfig
  DriveConfiguration/Segment:
    Shape = CIRCULAR
    SegmentReference = SEG_3_65
    StopReaction = UseAssemblySetting
    SpeedFilter = UseAssemblySetting
8F1I01.BB4B.xxxx-68 : 8F1I01.BB4B.xxxx-1 v1.0.0.1  [PLK1 -> 8F1I01.AB2B.xxxx-67.PLK2 (NodeNumber=68) [Cable Type=PowerlinkCable, Length=10, Version=1.0.0.2]; PLK2 -> 8F1I01.BB4B.xxxx-69.PLK1 (NodeNumber=68) [Cable Type=PowerlinkCable, Length=10, Version=1.0.0.2]]
  DriveConfiguration:
    McTypeID = LLMConfig
  DriveConfiguration/Segment:
    Shape = CIRCULAR
    SegmentReference = SEG_3_68
    StopReaction = UseAssemblySetting
    SpeedFilter = UseAssemblySetting
8F1I01.BB4B.xxxx-69 : 8F1I01.BB4B.xxxx-1 v1.0.0.1  [PLK1 -> 8F1I01.BB4B.xxxx-68.PLK2 (NodeNumber=69) [Cable Type=PowerlinkCable, Length=10, Version=1.0.0.2]; PLK2 -> 8F1I01.BB4B.xxxx-70.PLK1 (NodeNumber=69) [Cable Type=PowerlinkCable, Length=10, Version=1.0.0.2]; PLK3 -> X20HB2880c.ETH2 (NodeNumber=69) [Cable Type=PowerlinkCable, Length=10, Version=1.0.0.2]]
  DriveConfiguration:
    McTypeID = LLMConfig
  DriveConfiguration/Segment:
    Shape = CIRCULAR
    SegmentReference = SEG_3_69
    StopReaction = UseAssemblySetting
    SpeedFilter = UseAssemblySetting
8F1I01.BB4B.xxxx-70 : 8F1I01.BB4B.xxxx-1 v1.0.0.1  [PLK1 -> 8F1I01.BB4B.xxxx-69.PLK2 (NodeNumber=70) [Cable Type=PowerlinkCable, Length=10, Version=1.0.0.2]; PLK2 -> 8F1I01.BA2B.xxxx-71.PLK1 (NodeNumber=70) [Cable Type=PowerlinkCable, Length=10, Version=1.0.0.2]]
  DriveConfiguration:
    McTypeID = LLMConfig
  DriveConfiguration/Segment:
    Shape = CIRCULAR
    SegmentReference = SEG_3_70
    StopReaction = UseAssemblySetting
    SpeedFilter = UseAssemblySetting
8F1I01.BB4B.xxxx-73 : 8F1I01.BB4B.xxxx-1 v1.0.0.1  [PLK1 -> 8F1I01.AB2B.xxxx-72.PLK2 (NodeNumber=73) [Cable Type=PowerlinkCable, Length=10, Version=1.0.0.2]]
  DriveConfiguration:
    McTypeID = LLMConfig
  DriveConfiguration/Segment:
    Shape = CIRCULAR
    SegmentReference = SEG_3_73
    StopReaction = UseAssemblySetting
    SpeedFilter = UseAssemblySetting
8F1I01.BB4B.xxxx-74 : 8F1I01.BB4B.xxxx-1 v1.0.0.1  [PLK2 -> 8F1I01.BB4B.xxxx-75.PLK1 (NodeNumber=74) [Cable Type=PowerlinkCable, Length=10, Version=1.0.0.2]]
  DriveConfiguration:
    McTypeID = LLMConfig
  DriveConfiguration/Segment:
    Shape = CIRCULAR
    SegmentReference = SEG_2_74
    StopReaction = UseAssemblySetting
    SpeedFilter = UseAssemblySetting
8F1I01.BB4B.xxxx-75 : 8F1I01.BB4B.xxxx-1 v1.0.0.1  [PLK1 -> 8F1I01.BB4B.xxxx-74.PLK2 (NodeNumber=75) [Cable Type=PowerlinkCable, Length=10, Version=1.0.0.2]; PLK2 -> 8F1I01.BB4B.xxxx-76.PLK1 (NodeNumber=75) [Cable Type=PowerlinkCable, Length=10, Version=1.0.0.2]]
  DriveConfiguration:
    McTypeID = LLMConfig
  DriveConfiguration/Segment:
    Shape = CIRCULAR
    SegmentReference = SEG_2_75
    StopReaction = UseAssemblySetting
    SpeedFilter = UseAssemblySetting
8F1I01.BB4B.xxxx-76 : 8F1I01.BB4B.xxxx-1 v1.0.0.1  [PLK1 -> 8F1I01.BB4B.xxxx-75.PLK2 (NodeNumber=76) [Cable Type=PowerlinkCable, Length=10, Version=1.0.0.2]; PLK2 -> 8F1I01.BA2B.xxxx-77.PLK1 (NodeNumber=76) [Cable Type=PowerlinkCable, Length=10, Version=1.0.0.2]]
  DriveConfiguration:
    McTypeID = LLMConfig
  DriveConfiguration/Segment:
    Shape = CIRCULAR
    SegmentReference = SEG_2_76
    StopReaction = UseAssemblySetting
    SpeedFilter = UseAssemblySetting
8F1I01.BB4B.xxxx-79 : 8F1I01.BB4B.xxxx-1 v1.0.0.1  [PLK1 -> 8F1I01.AB2B.xxxx-78.PLK2 (NodeNumber=79) [Cable Type=PowerlinkCable, Length=10, Version=1.0.0.2]; PLK2 -> 8F1I01.BB4B.xxxx-80.PLK1 (NodeNumber=79) [Cable Type=PowerlinkCable, Length=10, Version=1.0.0.2]; PLK3 -> X20HB2880b.ETH1 (NodeNumber=79) [Cable Type=PowerlinkCable, Length=10, Version=1.0.0.2]]
  DriveConfiguration:
    McTypeID = LLMConfig
  DriveConfiguration/Segment:
    Shape = CIRCULAR
    SegmentReference = SEG_2_79
    StopReaction = UseAssemblySetting
    SpeedFilter = UseAssemblySetting
8F1I01.BB4B.xxxx-80 : 8F1I01.BB4B.xxxx-1 v1.0.0.1  [PLK1 -> 8F1I01.BB4B.xxxx-79.PLK2 (NodeNumber=80) [Cable Type=PowerlinkCable, Length=10, Version=1.0.0.2]; PLK2 -> 8F1I01.BB4B.xxxx-81.PLK1 (NodeNumber=80) [Cable Type=PowerlinkCable, Length=10, Version=1.0.0.2]]
  DriveConfiguration:
    McTypeID = LLMConfig
  DriveConfiguration/Segment:
    Shape = CIRCULAR
    SegmentReference = SEG_2_80
    StopReaction = UseAssemblySetting
    SpeedFilter = UseAssemblySetting
8F1I01.BB4B.xxxx-81 : 8F1I01.BB4B.xxxx-1 v1.0.0.1  [PLK1 -> 8F1I01.BB4B.xxxx-80.PLK2 (NodeNumber=81) [Cable Type=PowerlinkCable, Length=10, Version=1.0.0.2]; PLK2 -> 8F1I01.BA2B.xxxx-82.PLK1 (NodeNumber=81) [Cable Type=PowerlinkCable, Length=10, Version=1.0.0.2]]
  DriveConfiguration:
    McTypeID = LLMConfig
  DriveConfiguration/Segment:
    Shape = CIRCULAR
    SegmentReference = SEG_2_81
    StopReaction = UseAssemblySetting
    SpeedFilter = UseAssemblySetting
X20BB82 : X20BB82 v1.0.2.0
  Connector IF1:
    CycleTime = 10000
    BusLength = 50
    Stations = 32
    AsyncPayload = 96
X20BB82a : X20BB82 v1.0.2.0
  Connector IF1:
    CycleTime = 10000
    BusLength = 50
    Stations = 32
    AsyncPayload = 96
X20BC8083 : X20BC8083 v2.9.0.0  [PLK1 -> 5LS182.6-2.IF1 (NodeNumber=50) [Cable Type=PowerlinkCable, Length=10, Version=1.0.0.2]; PLK2 -> 8F1I01.BA2B.xxxx-53.PLK3 (NodeNumber=50) [Cable Type=PowerlinkCable, Length=10, Version=1.0.0.2]; SL -> X20BB82.SL1]
  Supervision = off
X20BC8083a : X20BC8083 v2.9.0.0  [PLK1 -> 5LS182.6-2.PLK2 (NodeNumber=10) [Cable Type=PowerlinkCable, Length=10, Version=1.0.0.2]; PLK2 -> 8F1I01.BB4B.xxxx-13.PLK3 (NodeNumber=10) [Cable Type=PowerlinkCable, Length=10, Version=1.0.0.2]; SL -> X20BB82a.SL1]
  Supervision = off
X20BM11 : X20BM11 v1.0.0.1  [X2X1 -> X20BB82.IF1]
X20BM11a : X20BM11 v1.0.0.1  [X2X1 -> X20BB82a.IF1]
X20BT9400 : X20BT9400 v1.0.2.0  [SS1 -> X20TB12b.SS; SL -> X20BM11.SL1]
  Supervision = off
  PowerInfo = on
X20BT9400a : X20BT9400 v1.0.2.0  [SS1 -> X20TB12c.SS; SL -> X20BM11a.SL1]
  Supervision = off
  PowerInfo = on
X20HB2880 : X20HB2880 v1.1.0.0  [ETH1 -> 8F1I01.AA66.xxxx-33.PLK3 [Cable Type=PowerlinkCable, Length=10, Version=1.0.0.2]; ETH2 -> 8F1I01.AB2B.xxxx-37.PLK3 [Cable Type=PowerlinkCable, Length=10, Version=1.0.0.2]; SS -> X20BB82a.SS2]
X20HB2880a : X20HB2880 v1.1.0.0  [ETH1 -> 8F1I01.AA66.xxxx-19.PLK3 [Cable Type=PowerlinkCable, Length=10, Version=1.0.0.2]; ETH2 -> 8F1I01.BA2B.xxxx-28.PLK3 [Cable Type=PowerlinkCable, Length=10, Version=1.0.0.2]; SS -> X20BB82a.SS1]
X20HB2880b : X20HB2880 v1.1.0.0  [ETH1 -> 8F1I01.BB4B.xxxx-79.PLK3 [Cable Type=PowerlinkCable, Length=10, Version=1.0.0.2]; ETH2 -> epl_icn.PLK1 [Cable Type=PowerlinkCable, Length=10, Version=1.0.0.2]; SS -> X20BB82.SS2]
X20HB2880c : X20HB2880 v1.1.0.0  [ETH1 -> 8F1I01.BA2B.xxxx-59.PLK3 [Cable Type=PowerlinkCable, Length=10, Version=1.0.0.2]; ETH2 -> 8F1I01.BB4B.xxxx-69.PLK3 [Cable Type=PowerlinkCable, Length=10, Version=1.0.0.2]; SS -> X20BB82.SS1]
X20PS9400 : X20PS9400 v1.0.2.4  [SS1 -> X20TB12.SS; PS -> X20BB82.PS1]
  Supervision = off
  PowerInfo = on
X20PS9400a : X20PS9400 v1.0.2.4  [SS1 -> X20TB12a.SS; PS -> X20BB82a.PS1]
  Supervision = off
  PowerInfo = on
X20TB12 : X20TB12 v1.0.0.0
X20TB12a : X20TB12 v1.0.0.0
X20TB12b : X20TB12 v1.0.0.0
X20TB12c : X20TB12 v1.0.0.0
epl_icn : epl_icn v1.3.2.0  [PLK1 -> X20HB2880b.ETH2 (NodeNumber=200) [Cable Type=PowerlinkCable, Length=10, Version=1.0.0.2]]
  RefConfiguration = Safety
  RefInterface = X20CP0484.IF3
```

### Cpu.per - 5PC900_TS17_00/Cpu.per
```iecst
VAR_CONFIG
	gTrack1 AT %M0; (* *)
	gTrack2 AT %M200; (* *)
	gTrack3 AT %M400; (* *)
	gTrack4 AT %M600; (* *)
	gTrack5 AT %M800; (* *)
	gTrack6 AT %M1000; (* *)
END_VAR
```

### Config_1.assembly - 5PC900_TS17_00/mappMotion/Config_1.assembly
```
Element gAssembly_1 (Type=assembly)
  Tracks:
    TrackSeparation = 0.030
    Track[1]:
      Segments:
        SegmentRef[1] = ::SEG_1_11
        SegmentRef[2] = ::SEG_1_12
        SegmentRef[3] = ::SEG_1_13
        SegmentRef[4] = ::SEG_1_14
        SegmentRef[5] = ::SEG_1_15
        SegmentRef[6] = ::SEG_1_16
        SegmentRef[7] = ::SEG_1_17
        SegmentRef[8] = ::SEG_1_18
        SegmentRef[9] = ::SEG_1_19
        SegmentRef[10] = ::SEG_1_20
        SegmentRef[11] = ::SEG_1_21
        SegmentRef[12] = ::SEG_1_22
        SegmentRef[13] = ::SEG_1_23
        SegmentRef[14] = ::SEG_1_24
        SegmentRef[15] = ::SEG_1_25
        SegmentRef[16] = ::SEG_1_26
        SegmentRef[17] = ::SEG_1_27
        SegmentRef[18] = ::SEG_1_28
        SegmentRef[19] = ::SEG_1_29
        SegmentRef[20] = ::SEG_1_30
        SegmentRef[21] = ::SEG_1_31
        SegmentRef[22] = ::SEG_1_32
        SegmentRef[23] = ::SEG_1_33
        SegmentRef[24] = ::SEG_1_34
        SegmentRef[25] = ::SEG_1_35
        SegmentRef[26] = ::SEG_1_36
      Position = Absolute
        SegmentRef = ::SEG_1_21
        SegmentCountDirection = RightToLeft
        Translation:
          X = 0.0
          Y = 0.0
          Z = 0.0
        Orientation:
          Angle1 = 0.0
          Angle2 = 0.0
          Angle3 = 0
    Track[2]:
      Segments:
        SegmentRef[1] = ::SEG_2_74
        SegmentRef[2] = ::SEG_2_75
        SegmentRef[3] = ::SEG_2_76
        SegmentRef[4] = ::SEG_2_77
        SegmentRef[5] = ::SEG_2_78
        SegmentRef[6] = ::SEG_2_79
        SegmentRef[7] = ::SEG_2_80
        SegmentRef[8] = ::SEG_2_81
        SegmentRef[9] = ::SEG_2_82
        SegmentRef[10] = ::SEG_2_83
      Position = RelativeToOne
        TrackSegmentPosition:
          SegmentRef = ::SEG_2_77
          PositionRelativeTo = FromEnd
        Base:
          SegmentRef = ::SEG_1_29
          Position = 0.321
    Track[3]:
      Segments:
        SegmentRef[1] = ::SEG_3_64
        SegmentRef[2] = ::SEG_3_65
        SegmentRef[3] = ::SEG_3_66
        SegmentRef[4] = ::SEG_3_67
        SegmentRef[5] = ::SEG_3_68
        SegmentRef[6] = ::SEG_3_69
        SegmentRef[7] = ::SEG_3_70
        SegmentRef[8] = ::SEG_3_71
        SegmentRef[9] = ::SEG_3_72
        SegmentRef[10] = ::SEG_3_73
      Position = RelativeToOne
        TrackSegmentPosition:
          SegmentRef = ::SEG_3_66
          PositionRelativeTo = FromEnd
        Base:
          SegmentRef = ::SEG_1_34
          Position = 0.33
    Track[4]:
      Segments:
        SegmentRef[1] = ::SEG_4_54
        SegmentRef[2] = ::SEG_4_55
        SegmentRef[3] = ::SEG_4_56
        SegmentRef[4] = ::SEG_4_57
        SegmentRef[5] = ::SEG_4_58
        SegmentRef[6] = ::SEG_4_59
        SegmentRef[7] = ::SEG_4_60
        SegmentRef[8] = ::SEG_4_61
        SegmentRef[9] = ::SEG_4_62
        SegmentRef[10] = ::SEG_4_63
      Position = RelativeToOne
        TrackSegmentPosition:
          SegmentRef = ::SEG_4_59
          PositionRelativeTo = FromEnd
        Base:
          SegmentRef = ::SEG_1_19
          Position = 0.33
    Track[5]:
      Segments:
        SegmentRef[1] = ::SEG_5_37
        SegmentRef[2] = ::SEG_5_38
        SegmentRef[3] = ::SEG_5_39
      Position = RelativeToOne
        TrackSegmentPosition:
          SegmentRef = ::SEG_5_39
          PositionRelativeTo = FromEnd
        Base:
          SegmentRef = ::SEG_1_11
    Track[6]:
      Segments:
        SegmentRef[1] = ::SEG_6_51
        SegmentRef[2] = ::SEG_6_52
        SegmentRef[3] = ::SEG_6_53
      Position = RelativeToOne
        TrackSegmentPosition:
          SegmentRef = ::SEG_6_51
        Base:
          SegmentRef = ::SEG_1_15
          PositionRelativeTo = FromEnd
  CommonSegmentSettings:
    SegmentSimulationOnPLC = Off
    StopReaction = InductionHalt
    SpeedFilter = Lowpass
      FilterTime = 0.0004
    ControllerParameters:
      DefaultParameter:
        Controller:
          Position:
            ProportionalGain = 160.0
          Speed:
            ProportionalGain = 80.0
            IntegrationTime = 0.0
          FeedForward:
            TotalMass = 1
            ForcePositive = 0.0
            ForceNegative = 0.0
            SpeedForceFactor = 0.0
            ForceLoad = 0.0
        MovementErrorLimits:
          PositionError = 1.0
          VelocityError = 10.0
      AdditionalParameterSets = NotUsed
  Shuttles:
    MaxShuttleCount = 50
    ShuttleStereotypes:
      ShuttleStRef[1] = ShuttleStereotype_1
    MagnetPlateConfigurations:
      ShuttleType[1] = 8F1SA.102.xxxxxx-x
    CollisionAvoidance:
      Strategy = Constant
      MaximumModelDimensions:
        Length:
          ExtentToFront = 0.2
          ExtentToBack = 0.2
        Width:
          Width = 0.2
  AssemblyFeatures:
    AssemblyFeatureRef[1] = AssemblyFeature_1
    AssemblyFeatureRef[2] = AssemblyFeature_2
  Visualization:
    MonitoringPv = ::gShuttleMon
    ProcessingTaskClass = 1
```

### Config_2.shuttlestereotype - 5PC900_TS17_00/mappMotion/Config_2.shuttlestereotype
```
Element ShuttleStereotype_1 (Type=shuttlestereotype)
  MeasurementUnit = 5067858
  MeasurementResolution = 0.000001
  MovementLimits = Internal
    VelocityIsReadOnly = 0
    Velocity:
      Velocity = 4
    AccelerationIsReadOnly = 0
    Acceleration:
      Acceleration = 40.0
    DecelerationIsReadOnly = 0
    Deceleration:
      Deceleration = 40.0
  JerkFilter = NotUsed
  UserData:
    Size = 12
  CollisionAvoidance:
    InitialModelDimensions = UseExplicitValues
      Length:
        ExtentToFront = 0.075
        ExtentToBack = 0.075
      Width:
        Width = 0.150
```

### Config_3.sector - 5PC900_TS17_00/mappMotion/Config_3.sector
```
Element SectorTrack1 (Type=sector)
  Type = Composed
    StartSegment:
      SegmentRef = ::SEG_1_11
    IntermediateSegments:
      SegmentRef[1] = ::SEG_1_12
      SegmentRef[2] = ::SEG_1_13
      SegmentRef[3] = ::SEG_1_14
      SegmentRef[4] = ::SEG_1_15
      SegmentRef[5] = ::SEG_1_16
      SegmentRef[6] = ::SEG_1_17
      SegmentRef[7] = ::SEG_1_18
      SegmentRef[8] = ::SEG_1_19
      SegmentRef[9] = ::SEG_1_20
      SegmentRef[10] = ::SEG_1_21
      SegmentRef[11] = ::SEG_1_22
      SegmentRef[12] = ::SEG_1_23
      SegmentRef[13] = ::SEG_1_24
      SegmentRef[14] = ::SEG_1_25
      SegmentRef[15] = ::SEG_1_26
      SegmentRef[16] = ::SEG_1_27
      SegmentRef[17] = ::SEG_1_28
      SegmentRef[18] = ::SEG_1_29
      SegmentRef[19] = ::SEG_1_30
      SegmentRef[20] = ::SEG_1_31
      SegmentRef[21] = ::SEG_1_32
      SegmentRef[22] = ::SEG_1_33
      SegmentRef[23] = ::SEG_1_34
      SegmentRef[24] = ::SEG_1_35
    EndSegment:
      SegmentRef = ::SEG_1_36
      PositionRelativeTo = FromEnd
Element SectorTrack2 (Type=sector)
  Type = Composed
    StartSegment:
      SegmentRef = ::SEG_2_74
    IntermediateSegments:
      SegmentRef[1] = ::SEG_2_75
      SegmentRef[2] = ::SEG_2_76
      SegmentRef[3] = ::SEG_2_77
      SegmentRef[4] = ::SEG_2_78
      SegmentRef[5] = ::SEG_2_79
      SegmentRef[6] = ::SEG_2_80
      SegmentRef[7] = ::SEG_2_81
      SegmentRef[8] = ::SEG_2_82
    EndSegment:
      SegmentRef = ::SEG_2_83
      PositionRelativeTo = FromEnd
Element SectorTrack5 (Type=sector)
  Type = Composed
    StartSegment:
      SegmentRef = ::SEG_5_37
    IntermediateSegments:
      SegmentRef[1] = ::SEG_5_38
    EndSegment:
      SegmentRef = ::SEG_5_39
      PositionRelativeTo = FromEnd
Element SectorTrack3 (Type=sector)
  Type = Composed
    StartSegment:
      SegmentRef = ::SEG_3_64
    IntermediateSegments:
      SegmentRef[1] = ::SEG_3_65
      SegmentRef[2] = ::SEG_3_66
      SegmentRef[3] = ::SEG_3_67
      SegmentRef[4] = ::SEG_3_68
      SegmentRef[5] = ::SEG_3_69
      SegmentRef[6] = ::SEG_3_70
      SegmentRef[7] = ::SEG_3_71
      SegmentRef[8] = ::SEG_3_72
    EndSegment:
      SegmentRef = ::SEG_3_73
      PositionRelativeTo = FromEnd
Element SectorTrack4 (Type=sector)
  Type = Composed
    StartSegment:
      SegmentRef = ::SEG_4_54
    IntermediateSegments:
      SegmentRef[1] = ::SEG_4_55
      SegmentRef[2] = ::SEG_4_56
      SegmentRef[3] = ::SEG_4_57
      SegmentRef[4] = ::SEG_4_58
      SegmentRef[5] = ::SEG_4_59
      SegmentRef[6] = ::SEG_4_60
      SegmentRef[7] = ::SEG_4_61
      SegmentRef[8] = ::SEG_4_62
    EndSegment:
      SegmentRef = ::SEG_4_63
      PositionRelativeTo = FromEnd
Element SectorTrack6 (Type=sector)
  Type = Composed
    StartSegment:
      SegmentRef = ::SEG_6_53
      PositionRelativeTo = FromEnd
    IntermediateSegments:
      SegmentRef[1] = ::SEG_6_52
    EndSegment:
      SegmentRef = ::SEG_6_51
```

### Config_4.processpointlist - 5PC900_TS17_00/mappMotion/Config_4.processpointlist
```
Element ProcessPointList_Sector (Type=processpointlist)
  ProcessPoint[0]:
    Name = PP_Track1
    SectorRef = SectorTrack1
    Position = 6.45
    PositionRelativeTo = FromEnd
    TriggerEventBufferSize = 10
    BarrierFunctionality = On
  ProcessPoint[1]:
    Name = PP_Track2
    SectorRef = SectorTrack2
    Position = 0.45
    PositionRelativeTo = FromEnd
    TriggerEventBufferSize = 10
    BarrierFunctionality = On
  ProcessPoint[2]:
    Name = PP_Track3
    SectorRef = SectorTrack3
    Position = 0.69
    PositionRelativeTo = FromEnd
    TriggerEventBufferSize = 10
    BarrierFunctionality = On
  ProcessPoint[3]:
    Name = PP_Track4
    SectorRef = SectorTrack4
    Position = 0.45
    TriggerEventBufferSize = 10
    BarrierFunctionality = On
  ProcessPoint[4]:
    Name = PP_Track5
    SectorRef = SectorTrack5
    Position = 0.45
    TriggerEventBufferSize = 10
    BarrierFunctionality = On
  ProcessPoint[5]:
    Name = PP_Track6
    SectorRef = SectorTrack6
    Position = 0.45
    PositionRelativeTo = FromEnd
    TriggerEventBufferSize = 10
    BarrierFunctionality = On
Element ProcessPointList_Track1 (Type=processpointlist)
  ProcessPoint[0]:
    Name = PP_Pre_Track4
    SectorRef = SectorTrack1
    Position = 2.94
    TriggerEventBufferSize = 10
    BarrierFunctionality = Off
  ProcessPoint[1]:
    Name = PP_Pre_Track2
    SectorRef = SectorTrack1
    Position = 5.73
    PositionRelativeTo = FromEnd
    TriggerEventBufferSize = 10
    BarrierFunctionality = Off
  ProcessPoint[2]:
    Name = PP_Pre_Track3
    SectorRef = SectorTrack1
    Position = 1.98
    PositionRelativeTo = FromEnd
    TriggerEventBufferSize = 10
    BarrierFunctionality = Off
```

### Config_5.assemblyfeature - 5PC900_TS17_00/mappMotion/Config_5.assemblyfeature
```
Element AssemblyFeature_1 (Type=assemblyfeature)
  Type = InitShuttleSim
    InitShuttleSim[1]:
      SectorRef = SectorTrack1
      Orientation = Positive
      ShuttleDefinition = ShuttleSetDefinition
        StartPosition = 2.0
        NumberOfShuttles = 15
        DistnaceBetweenShuttles = 0.15
    InitShuttleSim[2]:
      SectorRef = SectorTrack2
      Orientation = Negative
      ShuttleDefinition = ShuttleSetDefinition
        StartPosition = 0.1
        NumberOfShuttles = 5
        DistnaceBetweenShuttles = 0.15
    InitShuttleSim[3]:
      SectorRef = SectorTrack3
      Orientation = Negative
      ShuttleDefinition = ShuttleSetDefinition
        StartPosition = 0.1
        NumberOfShuttles = 5
        DistnaceBetweenShuttles = 0.15
    InitShuttleSim[4]:
      SectorRef = SectorTrack4
      Orientation = Negative
      ShuttleDefinition = ShuttleSetDefinition
        StartPosition = 0.1
        NumberOfShuttles = 5
        DistnaceBetweenShuttles = 0.15
    InitShuttleSim[5]:
      SectorRef = SectorTrack6
      Orientation = Positive
      ShuttleDefinition = ShuttleSetDefinition
        StartPosition = 0.1
        NumberOfShuttles = 3
        DistnaceBetweenShuttles = 0.15
Element AssemblyFeature_2 (Type=assemblyfeature)
  Type = ShtSectorAutoAttach
    Priority[1]:
      SectorRef = SectorTrack1
      Orientation = KeepSegment
    Priority[2]:
      SectorRef = SectorTrack2
      Orientation = KeepSegment
    Priority[3]:
      SectorRef = SectorTrack3
      Orientation = KeepSegment
    Priority[4]:
      SectorRef = SectorTrack4
      Orientation = KeepSegment
    Priority[5]:
      SectorRef = SectorTrack5
      Orientation = KeepSegment
    Priority[6]:
      SectorRef = SectorTrack6
      Orientation = KeepSegment
```

## Logical view

Binary libraries used (declarations not repeated): operator, runtime, astime, AsIecCon, AsZip, FileIO, brsystem, AsSem, sys_lib, AsBrStr, AsIODiag, DataObj, AsXml, standard, MpAlarmX, MpBase, MpAxis, McAxis, McBase, McAcpAx, McAcpTrak, CoTrace 5.09.0

### Global.var - Global variables
```iecst
(*shuttle-UserData structure*)
VAR
	testbutton : BOOL;
	gShuttleUserData : ShuttleUserData_typ;
END_VAR
```

- AcpTrakBasis_Visio.vsdx (binary file, 281912 bytes)
- AS4_HW_8YF1I01.AA66.00-1.exe (binary file, 153681 bytes)
- AS4_HW_8YF1I01.BA2B.00-1.exe (binary file, 158935 bytes)
- AS4_HW_8YF1I01.BB4B.00-1.exe (binary file, 157579 bytes)
### Library Logical/Libraries/brdkMU (ANSIC, version 5.00.0) - BRDK machine unit library. Provides functionality to control machines.
Depends on: AsSem, sys_lib, brsystem, brdkSTR

#### brdkEM.typ - brdkEM data types.
```iecst
TYPE
	brdk_em_states_typ :
		( (*Module states. Based on ISA–TR88.00.02 state model.*)
		STATE_DEACTIVATED := 0, (*State Type: Wait
The module has not been activated yet. An activate command will cause an exit from
DEACTIVATED to a ACTIVATING state.*)
		STATE_CLEARING := 1, (*State Type: Acting
Initiated by a state command to clear faults that may have occurred
when ABORTING, and are present in the ABORTED state before
proceeding to a STOPPED state.*)
		STATE_STOPPED := 2, (*State Type: Wait
The machine is powered and stationary after completing the
STOPPING state. All communications with other systems are
functioning (if applicable). A Reset command will cause an exit from
STOPPED to the RESETTING state.*)
		STATE_STARTING := 3, (*State Type: Acting
This state provides the steps needed to start the machine and is a
result of a starting type command (local or remote). Following this
command the machine will begin to Execute.*)
		STATE_IDLE := 4, (*State Type: Wait
This is a state which indicates that RESETTING is complete. This
state maintains the machine conditions which were achieved during
the RESETTING state, and performs operations required when the
machine is in IDLE.*)
		STATE_SUSPENDED := 5, (*State Type: Wait
The machine may be running at a relevant set point speed, but
there is no product being produced while the machine is waiting for
external process conditions to return to normal. When the offending
process conditions return to normal, the SUSPENDED state will
transition to UNSUSPENDING and hence continue towards the
normal EXECUTE state.*)
		STATE_EXECUTE := 6, (*State Type: Dual
Once the machine is processing materials it is deemed to be
executing or in the EXECUTE state. Different machine modes will
result in specific types of EXECUTE activities. For example, if the
machine is in the Production mode, the EXECUTE will result in
products being produced, while in Clean Out mode the EXECUTE
state refers to the action of cleaning the machine.*)
		STATE_STOPPING := 7, (*State Type: Acting
This state executes the logic which brings the machine to a
controlled stop as reflected by the STOPPED state. Normal
STARTING of the machine can not be initiated unless RESETTING
had taken place.*)
		STATE_ABORTING := 8, (*State Type: Acting
The ABORTED state can be entered at any time in response to the
Abort command or on the occurrence of a machine fault. The
aborting logic will bring the machine to a rapid safe stop. Operation
of the emergency stop will cause the machine to be tripped by its
safety system. It will also provide a signal to initiate the
ABORTING State.*)
		STATE_ABORTED := 9, (*State Type: Wait
This state maintains machine status information relevant to the
Abort condition. The machine can only exit the ABORTED state
after an explicit Clear command, subsequently to manual
intervention to correct and reset the detected machine faults.*)
		STATE_HOLDING := 10, (*State Type: Acting
When the machine is in the EXECUTE state, the Hold command
can be used to start HOLDING logic which brings the machine to a
controlled stop or to a state which represents HELD for the
particular unit control mode. A machine can go into this state either
when an internal equipment fault is automatically detected or by an
operator command. The Hold command offers the operator a safe
way to intervene manually in the process (such as removing a
broken bottle from the in-feed) and restarting execution when
conditions are safe. To be able to restart production correctly after
the HELD state, all relevant process set-points and return status of
the procedures at the time of receiving the Hold command must be
saved in the machine controller when executing the HOLDING
procedure.*)
		STATE_HELD := 11, (*State Type: Wait
The HELD state holds the machine's operation while material
blockages are cleared, or to stop throughput while a downstream
problem is resolved, or enable the safe correction of an equipment
fault before the production may be resumed.*)
		STATE_UNHOLDING := 12, (*State Type: Acting
The UNHOLDING state is a response to an Operator command to
resume the EXECUTE state. Issuing the Unhold command will
retrieve the saved set-points and return the status conditions to
prepare the machine to re-enter the normal EXECUTE state.*)
		STATE_SUSPENDING := 13, (*State Type: Acting
This state is a result of a change in monitored conditions due to
process conditions or factors. The trigger event will cause a
temporary suspension of the EXECUTE state. SUSPENDING is
typically the result of starvation of upstream material in-feeds (i.e.,
container feed, beverage feed, crown feed, lubricant feed, etc.) that
is outside the dynamic speed control range or a downstream outfeed
blockage that prevents the machine from EXECUTING
continued steady production. During the controlled sequence of
SUSPENDING the machine will transition to a SUSPENDED state.
The SUSPENDING state might be forced by the operator.*)
		STATE_UNSUSPENDING := 14, (*State Type: Acting
This state is a result of a machine generated request from
SUSPENDED state to go back to the EXECUTE state. The actions
of this state may include ramping up speeds, turning on vacuums,
and the re-engagement of clutches. This state is done prior to
EXECUTE state, and prepares the machine for the EXECUTE state.*)
		STATE_RESETTING := 15, (*State Type: Acting
This state is the result of a RESET command from the STOPPED or
complete state. RESETTING will typically cause a machine to
sound a horn and place the machine in a state where components
are energized awaiting a START command.*)
		STATE_COMPLETING := 16, (*State Type: Acting
This state is an automatic response from the EXECUTE state.
Normal operation has run to completion (i.e., processing of material
at the infeed will stop).*)
		STATE_COMPLETE := 17, (*State Type: Wait
The machine has finished the COMPLETING state and is now
waiting for a Reset command before transitioning to the
RESETTING state.*)
		STATE_DEACTIVATING := 18, (*State Type: Acting
This state is the result of a disabled ACTIVATE command.*)
		STATE_ACTIVATING := 19 (*State Type: Acting
State between DEACTIVATED and STOPPED. This state is done prior to
STOPPED state, and prepares the machine for the STOPPED state.*)
		) := STATE_DEACTIVATED;
	brdk_em_activation_typ :
		( (*Type of activation of equipment module.*)
		BRDK_EM_ACTIVATE := 0, (*Activates the equipment module.*)
		BRDK_EM_DEACTIVATE := 1, (*Deactivated the equipment module.*)
		BRDK_EM_ACTIVATE_BY_PARENT := 2 (*Automatically follows it's parent activation.*)
		) := BRDK_EM_DEACTIVATE;
	brdk_em_command_typ : 	STRUCT  (*Equipment module commands. Based on ISATR88.00.02.*)
		abort : BOOL := FALSE; (*Abort --> Go to STATE_ABORTING - Can be set in all states.*)
		clear : BOOL := FALSE; (*Clear --> Go to STATE_STOPPING - Can only be set in STATE_ABORTED.*)
		stop : BOOL := FALSE; (*Stop --> Go to STATE_STOPPING - Can be set in all states.*)
		reset : BOOL := FALSE; (*Reset --> Go to STATE_RESETTING - Can only be set in STATE_STOPPED.*)
		start : BOOL := FALSE; (*Start --> Go to STATE_STARTING - Can only be set in STATE_IDLE, STATE_SUSPENDED, STATE_HELD.*)
		hold : BOOL := FALSE; (*Hold --> Go to STATE_HOLDING - Can only be set in STATE_EXECUTE.*)
		suspend : BOOL := FALSE; (*Suspend --> Go to STATE_SUSPENDING - Can only be set in STATE_EXECUTE.*)
		complete : BOOL := FALSE; (*Complete --> Go to STATE_COMPLETING - Can only be set in STATE_EXECUTE.*)
		sc : BOOL := FALSE; (*The State Complete indication within the Acting state procedure will cause a state transition to occur. Same functionality as subsuate = SC.*)
	END_STRUCT;
	brdk_em_setup_typ : 	STRUCT  (*Equipment module setup structure.*)
		name : STRING[BRDK_MU_NAME_STRING_SIZE]; (*Name of the module. If empty the name of the task will be given.*)
		nameIdx : DINT := -1; (*Index to be added to name. If -1 no index will be set.*)
		reactTo : brdk_em_setup_react_typ := BRDK_EM_REACT_TO_ALL; (*Indicates which parent state the module should react to.*)
		parent : brdk_mu_setup_module_typ; (*Parameters to setup a parent module.*)
		skipStopSC : BOOL := FALSE; (*When this parameter is set the module will stop even though is not in sub state SC.*)
		sibling : ARRAY[0..BRDK_MU_MAX_SIBLINGS]OF brdk_mu_setup_module_typ; (*List of siblings to a module.*)
		activation : brdk_em_activation_typ := BRDK_EM_ACTIVATE; (*Type of activation of equipment module.*)
		useSubstateSC : BOOL := FALSE; (*Enables the if substate is set to SC it will work as cmd.sc.*)
		restore : brdk_em_setup_restore_typ; (*Functionality to restore a module to it's state after a e.g. power failure.*)
		status : brdk_em_setup_status_typ; (*Enable or disable status functionality.*)
	END_STRUCT;
	brdk_em_setup_status_typ : 	STRUCT  (*Enable or disable status functionality.*)
		stateSubstateMode : BOOL := TRUE; (*State, sub state and mode strings.*)
		last : BOOL := TRUE; (*Last log entries.*)
		waitingFor : BOOL := TRUE; (*Waiting for.*)
		interruptedBy : BOOL := TRUE; (*interrupted by.*)
	END_STRUCT;
	brdk_em_setup_react_typ :
		( (*Indicates witch command/state the module should react to.*)
		BRDK_EM_REACT_TO_ALL := 0, (*Reacts to all states.*)
		BRDK_EM_REACT_TO_ABORT_AND_STOP := 1, (*Reacts only to abort and stop states.*)
		BRDK_EM_REACT_TO_ABORT_ONLY := 2, (*Reacts only to abort state.*)
		BRDK_EM_REACT_TO_STOP_ONLY := 3, (*Reacts only to stop state.*)
		BRDK_EM_REACT_TO_NONE := 4, (*Doesn't react to any state or mode change. Runs total independent. Equal to the old cmd.ignore.*)
		BRDK_EM_LISTEN_TO_ABORT_AND_STOP := 5, (*The module listen to it's parent aborting and stopping only. Parent don't react to the module.*)
		BRDK_EM_LISTEN_TO_ABORT_ONLY := 6, (*The module listen to it's parent aborting only. Parent don't react to the module.*)
		BRDK_EM_LISTEN_TO_STOP_ONLY := 7 (*The module listen to it's parent stopping only. Parent don't react to the module.*)
		) := BRDK_EM_REACT_TO_ALL;
	brdk_em_setup_restore_typ : 	STRUCT  (*Functionality to restore a module to it's state after a e.g. power failure.*)
		pRestoreStruct : REFERENCE TO brdk_em_restore_module_typ; (*Pointer to the restore structure. Must be defined directly in the task in order to make it retain/permanent.*)
		activate : BOOL := FALSE; (*Activates the storing of the module information in the restore structure. This is to avoid overwriting the restore information.*)
	END_STRUCT;
	brdk_em_status_typ : 	STRUCT  (*Equipment module status.*)
		state : STRING[21]; (*String representation of the state.*)
		substate : STRING[BRDK_MU_MAX_DESCRIPTION_STRING]; (*Can be set in the task to descripe what the module is doing in this substate.*)
		mode : STRING[21]; (*String representation of the mode.*)
		name : STRING[BRDK_MU_NAME_STRING_SIZE]; (*Name of the module. If empty the name of the task will be given.*)
		time : UDINT; (*[ms] Actual time spend in the current state.*)
		last : ARRAY[0..BRDK_MU_MAX_LAST_SIZE]OF STRING[43]; (*The last state and substate the module was in and the spend time.*)
		childCount : UDINT; (*How many children are registered.*)
		waitingFor : brdk_em_waiting_for_typ; (*Info: Which child the parent and the underlying modules are waiting for.*)
		interruptedBy : brdk_em_interrupted_by_typ; (*Info: Which child interruped the parent by going into STOPPING or ABORTING.*)
		color : brdk_em_color_typ; (*Color depending af the unit state.*)
		lightTree : brdk_em_status_light_tree_typ; (*Light tree indicating the status of the module.*)
		cycleTime : UDINT; (*[µsec] Cycle time of the modules's task.*)
		parent : brdk_mu_status_module_typ; (*Information about the parent.*)
		sibling : ARRAY[0..BRDK_MU_MAX_SIBLINGS]OF brdk_mu_status_module_typ; (*List of available siblings.*)
		unvalidatedCmd : BOOL; (*Indicates that the current state cannot accept the given command.*)
		unvalidatedMode : BOOL; (*Indicates that the current state cannot accept the given mode change. Modes can only be changed in STATE_STOPPED and in STATE_ACTIVATING. The status flag will be reset by a state change.*)
		sleeping : BOOL; (*Indicates that the module is sleeping meaning that the module is not being executed because a new instance is being transferred.*)
		level : UDINT; (*Level in the hierarchy. Parent is level 0.*)
	END_STRUCT;
	brdk_em_status_light_tree_typ : 	STRUCT  (*Light tree indicating the status of the module. The idea of the light tree status is that it can be mapped directly to an output module.*)
		red : BOOL := FALSE; (*Color red.*)
		yellow : BOOL := FALSE; (*Color yellow.*)
		blue : BOOL := FALSE; (*Color blue.*)
		green : BOOL := FALSE; (*Color green.*)
	END_STRUCT;
	brdk_em_color_typ :
		( (*Color to display the current state.*)
		GREY := 0, (*Wait State - Unit is disabled*)
		BLUE := 1, (*Wait State – A stable state used to identify that a Unit has achieved a defined set of
conditions. In such a state the Unit is holding or maintaining a status until transitioning
to an Acting state (White color). The unit is powered and stationary.*)
		WHITE := 2, (*Acting State – A state which represents some processing activity, for example ramping
up speed.
It implies the single or repeated execution of processing steps in a logical order, for a
finite time or until a specific condition has been reached, for example within the
Starting state the quality of the received data is checking, before raping up speed for
execution.*)
		GREEN := 3, (*Dual State - The Unit is in a stable acting state. The unit is running and drives are active
and the unit is producing.*)
		RED := 4, (*Wait state – A state which represents an error state on the Unit. In this state the Unit is
not producing, until the operator have managed to make a transition to the EXECUTING
state. The state holds the units operation in a safe environment, until the command
unhold are executed. For example a material blockage will move the unit into the HELD
state. The unit will leave the state HELD, when the operator have entered the unit,
removed the the bloackage, and enabled all safeguards and activated the Unhold
command.*)
		ORANGE := 5 (*Wait State – A state which represents an error state on the line and the Unit is running
at a relevant set point speed, but there is no product being produced while the unit is
waiting for external process conditions to return to normal. The unit will also enter this
state if the operator want to have a break.*)
		) := GREY;
	brdk_em_interrupted_by_typ : 	STRUCT  (*Tells which unit has interrupted the hierarchy into STATE_ABORTING or STATE_STOPPING.*)
		name : STRING[BRDK_MU_NAME_STRING_SIZE]; (*Name of the child that has interrupted the parent.*)
		state : brdk_em_states_typ := STATE_DEACTIVATED; (*State info.*)
		substate : UINT := 0; (*Substate info.*)
	END_STRUCT;
	brdk_em_waiting_for_typ : 	STRUCT  (*Tells which child module the hierarchy are waiting for. Can be that the modules are waiting for more children, but only one of them a shown at a time.*)
		name : STRING[BRDK_MU_NAME_STRING_SIZE]; (*Name of the child that the parent is waiting for.*)
		substate : STRING[BRDK_MU_MAX_DESCRIPTION_STRING]; (*Child substate.*)
	END_STRUCT;
	brdk_em_internal_typ : 	STRUCT  (*Internal variables.*)
		SemCreate_0 : SemCreate; (*Module semaphore.*)
		old : brdk_em_state_old_typ; (*Last state info.*)
		flashTime : UDINT := 0; (*Flash time counter.*)
		initSubstate : UINT := 0; (*Internal temp sub state to be used in STATE_DEACTIVATED.*)
		pInterrupter : UDINT := 0; (*Pointer to the module that interrupted.*)
		findParent : BOOL := FALSE; (*The module automatically finds it's parent's state.*)
		muList : brdk_em_internal_mu_list_typ; (*Holds index's in the MU list.*)
		cmdSC : BOOL; (*Internal command state complete.*)
		statusCnt : brdk_em_internal_status_cnt_typ; (*Status counter to indicate if a status change has been made.*)
		waitingForIdx : DINT := -1; (*Index of the module we are waiting for.*)
		deactivateRequest : BOOL := TRUE; (*A request to deactivate the mdule has been made.*)
	END_STRUCT;
	brdk_em_internal_status_cnt_typ : 	STRUCT  (*Status counter to indicate if a status change has been made.*)
		internalCounter : DINT := -1; (*Internal counter which will be incremented if the status changes.*)
		externalCounter : DINT := -1; (*External counter which will hold the status counter of the waiting for module.*)
	END_STRUCT;
	brdk_em_state_old_typ : 	STRUCT  (*Holds the old states.*)
		state : brdk_em_states_typ := STATE_DEACTIVATED; (*Old state.*)
		substate : UINT := 0; (*Old substate.*)
		mode : DINT := 0; (*Old mode.*)
		reactTo : brdk_em_setup_react_typ := BRDK_EM_REACT_TO_ALL; (*Old reactTo.*)
	END_STRUCT;
	brdk_em_internal_mu_list_typ : 	STRUCT  (*Holds index's in the MU list.*)
		idx : DINT := -1; (*Own index in the mu list.*)
		parentIdx : DINT := -1; (*Parent index in the mu list.*)
		siblingIdx : ARRAY[0..BRDK_MU_MAX_SIBLINGS]OF DINT := [4(-1)]; (*Siblings index in the mu list.*)
		childrenIdx : ARRAY[0..BRDK_EM_MAX_CHILDREN]OF DINT; (*Children index in the mu list.*)
	END_STRUCT;
	brdk_em_restore_module_typ : 	STRUCT  (*Hold information that can be used to restore to it's active state in the case of a power failure.*)
		state : brdk_em_states_typ; (*Restored state.*)
		substate : UINT; (*Restored sub state.*)
		sc : BOOL; (*Restores state complete.*)
		mode : UINT; (*Restore mode.*)
	END_STRUCT;
	brdk_em_static_status_text_typ :
		( (*Internal enum to set a static status text*)
		STATUS_TEXT_DESCRIPTION := 0,
		STATUS_TEXT_ACTIVATION := 1
		);
END_TYPE
```

#### brdkMU.var - brdkMU constants.
```iecst
VAR CONSTANT
	BRDK_MU_MAX_MODULES : UINT := 2000; (*Maximum numbers of machine units.*)
	BRDK_MU_NAME_STRING_SIZE : UINT := 80; (*Maximum size of the module name.*)
	BRDK_MU_MAX_DESCRIPTION_STRING : UINT := 200; (*Maximum size of string description.*)
	BRDK_MU_MAX_LAST_SIZE : UINT := 19; (*Maximum size of last/history array. (19 means 20)*)
	BRDK_MU_MAX_SIBLINGS : UINT := 3; (*Maximum number of siblings to a module. (3 means 4)*)
	BRDK_EM_MAX_CHILDREN : UINT := 99; (*Maximum number of children to a module.*)
	BRDK_EM_FLASH_TIME : UINT := 1000; (*[ms] Color flash time.*)
	BRDK_MU_MAX_TOP_MODULES : UINT := 20; (*Maximum number of top equipment modules. A top module is an equipment module with no parent.*)
	BRDK_UM_MAX_PRODUCTS : UINT := 9; (*Maximum number of product PackTags. (9 means 10)*)
	MODE_UNDEFINED : DINT := 0; (*Initialization of Unit when power up.*)
	MODE_PRODUCING : DINT := 1; (*This represents the mode which is utilized for routine production. The machine executes
relevant logic in response to commands which are either entered directly by the operator or
issued by another supervisory system.*)
	MODE_MAINTENANCE : DINT := 2; (*This mode may allow suitably authorized personnel the ability to run an individual machine
independent of other machines in a production line. This mode would typically be used for
faultfinding, machine trials, or testing operational improvements.*)
	MODE_MANUAL : DINT := 3; (*This provides direct control of individual machine modules. This feature is available
depending upon the mechanical constraints of the mechanisms being exercised. This feature
may be used for the commissioning of individual drives, verifying the operation of
synchronized drives, testing the drive as a result of modifying parameters, etc.*)
	MODE_CLEAN : DINT := 16; (*Clean the Unit.*)
	MODE_JOG : DINT := 17; (*Step through a process.*)
	MODE_CIP : DINT := 18; (*Cleaning in progress.*)
	MODE_CALIBRATING : DINT := 19; (*Calibrating mode.*)
	SC : UINT := 65000; (*Sub state completet state. If enable and substate is set to SC it will work as the cmd.sc.*)
END_VAR
```

#### brdkMU.fun - brdkMU functions.
```iecst
FUNCTION_BLOCK brdkEM (*Represents an equipment module.*) (*$GROUP=User*)
	VAR_INPUT
		description : STRING[BRDK_MU_MAX_DESCRIPTION_STRING]; (*Description of what the substate is doing or waiting for.*)
		mode : DINT := MODE_PRODUCING; (*Control modes. Based on ISA-TR88.00.02 control modes. Modes can only be changed in STATE_STOPPED.*)
		cmd : brdk_em_command_typ; (*Control commands. Based on ISA-TR88.00.02 commands.*)
		setup : brdk_em_setup_typ; (*Setup of module.*)
		substate : UINT := 0; (*Equipment module substate can be used in the task. When a state is done set cmd.sc = true and the fb will take the unit to it's next state.*)
	END_VAR
	VAR_OUTPUT
		state : brdk_em_states_typ := STATE_DEACTIVATED; (*Equipment module state. State changes are controlled in the fb and is not allowed outside this fb. Based on ISA-TR88.00.02 states.*)
		status : brdk_em_status_typ; (*Module status.*)
	END_VAR
	VAR
		internal : brdk_em_internal_typ; (*Internal variables.*)
	END_VAR
END_FUNCTION_BLOCK

FUNCTION brdkEMSleep : DINT (*Put an equipment module to sleep. $RETURN=index;Index in the list.*) (*$GROUP=User,$CAT=User,$GROUPICON=User.png,$CATICON=User.png*)
	VAR_INPUT
		pEM : UDINT; (*Pointer to the equipment module.*)
	END_VAR
END_FUNCTION

FUNCTION brdkEMModeToA : UDINT (*Converts an equipment module mode int to a string representation. $RETURN=pointer;String pointer to mode string.*) (*$GROUP=User,$CAT=User,$GROUPICON=User.png,$CATICON=User.png*)
	VAR_INPUT
		mode : DINT; (*Equipment module mode.*)
	END_VAR
END_FUNCTION

FUNCTION brdkEMStateToA : UDINT (*Converts an equipment module state enum to a string representation. $RETURN=pointer;String pointer to state string.*) (*$GROUP=User,$CAT=User,$GROUPICON=User.png,$CATICON=User.png*)
	VAR_INPUT
		state : brdk_em_states_typ; (*Equipment module state.*)
	END_VAR
END_FUNCTION

FUNCTION_BLOCK brdkCM (*Represents a control module. The module does not follow the ISA-TR88.00.02 standard.*) (*$GROUP=User,$CAT=User,$GROUPICON=User.png,$CATICON=User.png*)
	VAR_INPUT
		description : STRING[BRDK_MU_MAX_DESCRIPTION_STRING]; (*Description of what the state / substate is doing or waiting for.*)
		state : UINT := 0; (*Control module state must be used in the task.*)
		substate : UINT := 0; (*Control module substate must be used in the task.*)
		setup : brdk_cm_setup_typ; (*Setup of module.*)
	END_VAR
	VAR_OUTPUT
		status : brdk_cm_status_typ; (*Module status.*)
	END_VAR
	VAR
		internal : brdk_cm_internal_typ; (*Internal variables.*)
	END_VAR
END_FUNCTION_BLOCK

FUNCTION brdkCMSleep : DINT (*Put a control module to sleep. $RETURN=index;Index in the list.*) (*$GROUP=User,$CAT=User,$GROUPICON=User.png,$CATICON=User.png*)
	VAR_INPUT
		pCM : UDINT; (*Pointer to the control module.*)
	END_VAR
END_FUNCTION

FUNCTION brdkCMChangeParent : DINT (*Changes the parent of a control module. $RETURN=index;Index in the new parent.*) (*$GROUP=User,$CAT=User,$GROUPICON=User.png,$CATICON=User.png*)
	VAR_INPUT
		pCM : UDINT; (*Pointer to the control module.*)
		pParentName : UDINT; (*Pointert to the logical name of the parent module.*)
		parentIndex : DINT; (*Index to be added to the module name. If -1 no index will be set.*)
	END_VAR
END_FUNCTION

FUNCTION_BLOCK brdkUM (*Unit Machine / Information Receiver module. It makes communication with a remote system easy. This fb makes it possible to remote control an equipment module.*) (*$GROUP=User,$CAT=User,$GROUPICON=User.png,$CATICON=User.png*)
	VAR_INPUT
		mode : brdk_um_mode_typ := BRDK_UM_MODE_MANUAL; (*Communication mode.*)
		pEM : UDINT; (*Pointer to the main equipment module (machine unit).*)
		Status : brdk_um_pml_s_typ; (*Status tags.*)
		Admin : brdk_um_pml_a_typ; (*Administration tags.*)
	END_VAR
	VAR_OUTPUT
		Command : brdk_um_pml_c_typ; (*Command tags.*)
	END_VAR
	VAR
		internal : brdk_um_pml_internal_typ; (*Internal variables.*)
	END_VAR
END_FUNCTION_BLOCK
```

#### brdkEM.c - Represents an equipment module.
```c
#include <brdkEM_func.h>

void brdkEM(struct brdkEM* this) {

	brdkEM_typ* parent;
	wakeMU(this->internal.muList.idx,(unsigned long)this);
	parent = getEm(this->internal.muList.parentIdx);

	/* if enabled command state completet can be set by settings the sub state to SC (65000) */
	if(this->setup.useSubstateSC) this->internal.cmdSC = this->substate == SC ? true : this->cmd.sc;
	else this->internal.cmdSC = this->cmd.sc;

	/* update information about the last */

	switch(this->state) {

		case STATE_STOPPED:
			this->status.color = BLUE;
			lightTree(this,BLUE,RED);
			setSubStateText(this,0);
			observeChildrensState(this, 2, STATE_ABORTING, STATE_ABORTED);						/* check if a child is in STATE- ABORTING or ABORTED */
			observeParentState(this, parent, 2, STATE_RESETTING, STATE_ABORTING);					/* check if parent is in STATE- RESETTING */
			if(this->internal.findParent) findParent(this,parent,STATE_RESETTING,11,STATE_IDLE,STATE_STARTING,STATE_EXECUTE,STATE_HOLDING,STATE_HELD,STATE_UNHOLDING,STATE_SUSPENDING,STATE_SUSPENDED,STATE_UNSUSPENDING,STATE_COMPLETING,STATE_COMPLETE);
			checkCommands(this, parent, 3, STATE_RESETTING, STATE_ABORTING, STATE_DEACTIVATING);		/* check commands reset, abort, not activate */
			setChildrenMode(this);
			if(this->mode == MODE_UNDEFINED) this->mode = MODE_PRODUCING;
			this->status.level = parent != NULL ? parent->status.level+1  : 0;	/* sets the hierarchy level */
			break;

		case STATE_RESETTING:
			this->status.color = WHITE;
			lightTree(this,BLUE,WHITE);
			setSubStateText(this,0);
			checkChildren(this, STATE_IDLE); 													/* CHECK IF ALL CHILDREN ARE IN STATE_IDLE */
			observeChildrensState(this, 3, STATE_ABORTING, STATE_ABORTED, STATE_STOPPING);		/* CHECK IF ONE CHILD IS IN STATE_ABORTING OR STATE_ABORTED */
			observeParentState(this,parent, 2, STATE_STOPPING,STATE_ABORTING);							/* checks if parent is in STATE- STOPPING or ABORTING */
			checkCommands(this, parent, 2, STATE_STOPPING, STATE_ABORTING);								/* check commands stop and abort */
			break;

		case STATE_IDLE:
			this->status.color = BLUE;
			lightTree(this,BLUE,WHITE);
			setSubStateText(this,0);
			observeChildrensState(this, 4, STATE_ABORTING, STATE_ABORTED, STATE_STOPPING, STATE_STOPPED);		/* check child state */
			observeParentState(this, parent, 3,STATE_STARTING,STATE_STOPPING,STATE_ABORTING);						/* CHECK STATE OF THE PARENT AND MAYBE FOLLOW */
			if(this->internal.findParent) findParent(this,parent,STATE_STARTING,9,STATE_EXECUTE,STATE_HOLDING,STATE_HELD,STATE_UNHOLDING,STATE_SUSPENDING,STATE_SUSPENDED,STATE_UNSUSPENDING,STATE_COMPLETING,STATE_COMPLETE);
			checkCommands(this, parent, 3, STATE_STOPPING, STATE_ABORTING, STATE_STARTING);								/* check commands stop, abort, start */
			break;

		case STATE_STARTING:
			this->status.color = WHITE;
			lightTree(this,flashColor(this,GREEN),WHITE);
			setSubStateText(this,0);
			checkChildren(this, STATE_EXECUTE); 															/* SUBSTATE MUST BE IN SC - CHECK IF ALL CHILDREN ARE IN STATE_EXECUTE */
			observeChildrensState(this, 4, STATE_ABORTING, STATE_ABORTED, STATE_STOPPING, STATE_STOPPED);	/* CHECK IF ONE CHILD IS IN STATE */
			observeParentState(this, parent,2,STATE_STOPPING,STATE_ABORTING); 										/* CHECK STATE OF THE PARENT AND MAYBE FOLLOW */
			checkCommands(this, parent, 2, STATE_STOPPING, STATE_ABORTING);											/* check commands stop, abort */
			break;

		case STATE_EXECUTE:
			this->status.color = GREEN;
			lightTree(this,GREEN,WHITE);
			setSubStateText(this,0);
			observeChildrensState(this, 8, STATE_ABORTING, STATE_ABORTED, STATE_STOPPING, STATE_STOPPED, STATE_SUSPENDING, STATE_SUSPENDED, STATE_HOLDING, STATE_HELD);		/* CHECK IF ONE CHILD IS IN STATE */
			observeParentState(this,parent,5,STATE_HOLDING,STATE_SUSPENDING,STATE_COMPLETING,STATE_STOPPING,STATE_ABORTING); /* CHECK STATE OF THE PARENT AND MAYBE FOLLOW */
			if(this->internal.findParent) findParent(this,parent,STATE_EXECUTE,7,STATE_HOLDING,STATE_HELD,STATE_SUSPENDING,STATE_SUSPENDED,STATE_COMPLETING,STATE_COMPLETE);
			checkCommands(this, parent, 5, STATE_STOPPING, STATE_ABORTING, STATE_HOLDING, STATE_SUSPENDING, STATE_COMPLETING);		/* check commands stop, abort, hold, suspend, complete */
			break;

		case STATE_HOLDING:
			this->status.color = WHITE;
			lightTree(this,flashColor(this,RED),WHITE);
			setSubStateText(this,0);
			checkChildren(this, STATE_HELD); 											/* SUBSTATE MUST BE IN SC - CHECK IF ALL CHILDREN ARE IN STATE_EXECUTE */
			observeChildrensState(this, 2, STATE_ABORTING, STATE_ABORTED);				/* CHECK IF ONE CHILD IS IN STATE */
			observeParentState(this,parent,2,STATE_STOPPING,STATE_ABORTING); 					/* CHECK STATE OF THE PARENT AND MAYBE FOLLOW */
			checkCommands(this, parent, 2, STATE_STOPPING, STATE_ABORTING);						/* check commands stop, abort */
			break;

		case STATE_HELD:
			this->status.color = RED;
			lightTree(this,flashColor(this,RED),WHITE);
			setSubStateText(this,0);
			observeChildrensState(this, 2, STATE_ABORTING, STATE_ABORTED);					/* CHECK IF ONE CHILD IS IN STATE */
			observeParentState(this,parent,3,STATE_UNHOLDING,STATE_STOPPING,STATE_ABORTING); 	/* CHECK STATE OF THE PARENT AND MAYBE FOLLOW */
			if(this->internal.findParent) findParent(this,parent,STATE_UNHOLDING,6,STATE_EXECUTE,STATE_SUSPENDING,STATE_SUSPENDED,STATE_UNSUSPENDING,STATE_COMPLETING,STATE_COMPLETE);
			checkCommands(this, parent, 3, STATE_STOPPING, STATE_ABORTING, STATE_UNHOLDING);		/* check commands stop, abort, start */
			break;

		case STATE_UNHOLDING:
			this->status.color = WHITE;
			lightTree(this,RED,GREEN);
			setSubStateText(this,0);
			checkChildren(this, STATE_EXECUTE); 											/* SUBSTATE MUST BE IN SC - CHECK IF ALL CHILDREN ARE IN STATE_EXECUTE */
			observeChildrensState(this, 2, STATE_ABORTING, STATE_ABORTED);					/* CHECK IF ONE CHILD IS IN STATE */
			observeParentState(this,parent,2,STATE_STOPPING,STATE_ABORTING); 						/* CHECK STATE OF THE PARENT AND MAYBE FOLLOW */
			checkCommands(this, parent, 2, STATE_STOPPING, STATE_ABORTING);							/* check commands stop, abort */
			break;

		case STATE_SUSPENDING:
			this->status.color = WHITE;
			lightTree(this,ORANGE,WHITE);
			setSubStateText(this,0);
			checkChildren(this, STATE_SUSPENDED); 											/* SUBSTATE MUST BE IN SC - CHECK IF ALL CHILDREN ARE IN STATE_EXECUTE */
			observeChildrensState(this, 2, STATE_ABORTING, STATE_ABORTED);					/* CHECK IF ONE CHILD IS IN STATE */
			observeParentState(this,parent,2,STATE_STOPPING,STATE_ABORTING); 						/* CHECK STATE OF THE PARENT AND MAYBE FOLLOW */
			checkCommands(this, parent, 2, STATE_STOPPING, STATE_ABORTING);							/* check commands stop, abort */
			break;

		case STATE_SUSPENDED:
			this->status.color = ORANGE;
			lightTree(this,ORANGE,WHITE);
			setSubStateText(this,0);
			observeChildrensState(this, 2, STATE_ABORTING, STATE_ABORTED);					/* CHECK IF ONE CHILD IS IN STATE */
			observeParentState(this,parent,3,STATE_UNSUSPENDING,STATE_STOPPING,STATE_ABORTING); 	/* CHECK STATE OF THE PARENT AND MAYBE FOLLOW */
			if(this->internal.findParent) findParent(this,parent,STATE_UNSUSPENDING,6,STATE_EXECUTE,STATE_HOLDING,STATE_HELD,STATE_UNHOLDING,STATE_COMPLETING,STATE_COMPLETE);
			checkCommands(this, parent, 3, STATE_STOPPING, STATE_ABORTING, STATE_UNSUSPENDING);		/* check commands stop, abort, start */
			break;

		case STATE_UNSUSPENDING:
			this->status.color = WHITE;
			lightTree(this,ORANGE,GREEN);
			setSubStateText(this,0);
			checkChildren(this, STATE_EXECUTE); 											/* SUBSTATE MUST BE IN SC - CHECK IF ALL CHILDREN ARE IN STATE_EXECUTE */
			observeChildrensState(this, 2, STATE_ABORTING, STATE_ABORTED);					/* CHECK IF ONE CHILD IS IN STATE */
			observeParentState(this,parent,2,STATE_STOPPING,STATE_ABORTING); 						/* CHECK STATE OF THE PARENT AND MAYBE FOLLOW */
			checkCommands(this, parent, 2, STATE_STOPPING, STATE_ABORTING);							/* check commands stop, abort */
			break;

		case STATE_COMPLETING:
			this->status.color = WHITE;
			lightTree(this,GREEN,BLUE);
			setSubStateText(this,0);
			checkChildren(this, STATE_COMPLETE); 											/* SUBSTATE MUST BE IN SC - CHECK IF ALL CHILDREN ARE IN STATE_EXECUTE */
			observeChildrensState(this, 2, STATE_ABORTING, STATE_ABORTED);					/* CHECK IF ONE CHILD IS IN STATE */
			observeParentState(this,parent,2,STATE_STOPPING,STATE_ABORTING); 						/* CHECK STATE OF THE PARENT AND MAYBE FOLLOW */
			checkCommands(this, parent, 2, STATE_STOPPING, STATE_ABORTING);							/* check commands stop, abort */
			break;

		case STATE_COMPLETE:
			this->status.color = BLUE;
			lightTree(this,flashColor(this,BLUE),WHITE);
			setSubStateText(this,0);
			observeChildrensState(this, 2, STATE_ABORTING, STATE_ABORTED);					/* CHECK IF ONE CHILD IS IN STATE */
			observeParentState(this,parent,3,STATE_RESETTING,STATE_STOPPING,STATE_ABORTING); 		/* CHECK STATE OF THE PARENT AND MAYBE FOLLOW */
			if(this->internal.findParent) findParent(this,parent,STATE_RESETTING,10,STATE_IDLE,STATE_STARTING,STATE_EXECUTE,STATE_HOLDING,STATE_HELD,STATE_UNHOLDING,STATE_SUSPENDING,STATE_SUSPENDED,STATE_UNSUSPENDING,STATE_COMPLETING);
			checkCommands(this, parent, 3, STATE_STOPPING, STATE_ABORTING, STATE_RESETTING);		/* check commands stop, abort, reset */
			break;

		case STATE_ABORTING:
			this->status.color = WHITE;
			lightTree(this,RED,WHITE);
			setSubStateText(this,0);
			checkChildren(this, STATE_ABORTED);
			break;

		case STATE_ABORTED:
			this->status.color = RED;
			lightTree(this,RED,WHITE);
			setSubStateText(this,0);
			observeParentState(this,parent,1,STATE_CLEARING); 										/* CHECK STATE OF THE PARENT AND MAYBE FOLLOW */
			checkCommands(this, parent, 2, STATE_CLEARING, STATE_DEACTIVATING);						/* check commands clar, not activate */
			break;

		case STATE_CLEARING:
			this->status.color = WHITE;
			lightTree(this,RED,flashColor(this,BLUE));
			setSubStateText(this,0);
			checkChildren(this, STATE_STOPPED); 										/* SUBSTATE MUST BE IN SC - CHECK IF ALL CHILDREN ARE IN STATE_EXECUTE */
			observeChildrensState(this, 2, STATE_ABORTING, STATE_ABORTED);				/* CHECK IF ONE CHILD IS IN STATE */
			observeParentState(this,parent,2,STATE_STOPPING,STATE_ABORTING); 			/* CHECK STATE OF THE PARENT AND MAYBE FOLLOW */
			break;

		case STATE_STOPPING:
			this->status.color = WHITE;
			lightTree(this,GREEN,BLUE);
			setSubStateText(this,0);
			checkChildren(this, STATE_STOPPED); 									/* SUBSTATE MUST BE IN SC - CHECK IF ALL CHILDREN ARE IN STATE_EXECUTE */
			observeChildrensState(this, 2, STATE_ABORTING, STATE_ABORTED);			/* CHECK IF ONE CHILD IS IN STATE */
			observeParentState(this,parent,1,STATE_ABORTING); 								/* CHECK STATE OF THE PARENT AND MAYBE FOLLOW */
			checkCommands(this, parent, 2, STATE_ABORTING, STATE_DEACTIVATING);								/* check commands abort */
			break;

		case STATE_DEACTIVATING:
			this->status.color = WHITE;
			lightTree(this,flashColor(this,GREY),WHITE);
			setSubStateText(this,0);
			this->internal.initSubstate = 0;
			if(this->internal.cmdSC) {
				UnregisterChild(this, parent);
				this->state = STATE_DEACTIVATED;
			}
			break;

		case STATE_ACTIVATING:
			this->status.color = WHITE;
			lightTree(this,flashColor(this,GREY),BLUE);
			if(this->internal.cmdSC) {
				if(parent != NULL) {
					switch(parent->state) {

						case STATE_STOPPED:
							if(this->mode == MODE_UNDEFINED && this->setup.reactTo == BRDK_EM_REACT_TO_NONE) this->mode = MODE_PRODUCING;
							else this->mode = parent->mode;
							this->state = STATE_STOPPED;
							break;

						case STATE_DEACTIVATED:
							setSubStateText(this,(unsigned long)"waiting for parent to be activated");
							break;

						default:
							setSubStateText(this,(unsigned long)"waiting for parent to be in STATE_STOPPED");
							break;

					}
				}
				else {
					if(this->mode == MODE_UNDEFINED) this->mode = MODE_PRODUCING;
					this->state = STATE_STOPPED;
				}
			setSubStateText(this,0);
			}
			break;

		case STATE_DEACTIVATED:
			this->status.color = GREY;
			lightTree(this,GREY,WHITE);
			setSubStateText(this, 0);
			if(this->status.cycleTime == 0) this->status.cycleTime = getCycleTime();								/* get the modules cycle time */
			brdkEMInitialize(this,parent);
			checkCommands(this, parent, 1, STATE_ACTIVATING);
			break;
	}

	/* mode change */
	if(this->mode != this->internal.old.mode) {
		if(this->state == STATE_STOPPED || this->state == STATE_ACTIVATING || this->state == STATE_DEACTIVATING || this->state == STATE_DEACTIVATED) {
			/* save last state for log */
			if(this->setup.status.last) {
				brdkStrMemMove((unsigned long)this->status.last[1],(unsigned long)this->status.last[0], sizeof(this->status.last[0])*BRDK_MU_MAX_LAST_SIZE);
				brdkStrCpy((unsigned long)this->status.last[0], brdkEMModeToA(this->internal.old.mode));
				brdkStrCat((unsigned long)this->status.last[0], (unsigned long)"-->");
				brdkStrCat((unsigned long)this->status.last[0], brdkEMModeToA(this->mode));
			}
			this->internal.old.mode = this->mode;
			if(this->setup.status.stateSubstateMode) brdkStrCpy((unsigned long)this->status.mode,brdkEMModeToA(this->mode));
		}
		else { /* avoid mode being change in other states than STATE_STOPPED */
			this->status.unvalidatedMode = true;
			this->mode = this->internal.old.mode;
		}
	}

	this->status.time += this->status.cycleTime/1000;

	/* state change */
	if(this->state != this->internal.old.state || this->substate != this->internal.old.substate) {
		/* save last state for log */
		if(this->setup.status.last) {
			brdkStrMemMove((unsigned long)this->status.last[1],(unsigned long)this->status.last[0], sizeof(this->status.last[0])*BRDK_MU_MAX_LAST_SIZE);
			brdkStrCpy((unsigned long)this->status.last[0],(unsigned long)this->status.state);
			brdkStrCat((unsigned long)this->status.last[0],(unsigned long)": ");
			if(this->state != this->internal.old.state) brdkStrAppendUdintToA(this->substate,(unsigned long)this->status.last[0],BRDK_STR_CONVERT_DECIMAL,-1);
			else brdkStrAppendUdintToA(this->internal.old.substate,(unsigned long)this->status.last[0],BRDK_STR_CONVERT_DECIMAL,-1);
			brdkStrCat((unsigned long)this->status.last[0],(unsigned long)": ");
			brdkStrAppendUdintToA(this->status.time,(unsigned long)this->status.last[0],BRDK_STR_CONVERT_DECIMAL,-1);
			brdkStrCat((unsigned long)this->status.last[0],(unsigned long)"ms");
		}
		if(this->setup.status.stateSubstateMode) brdkStrCpy((unsigned long)this->status.state,(unsigned long)brdkEMStateToA(this->state));
		if(this->state != this->internal.old.state) {
			/* log who interrupted the module */
			if(this->internal.pInterrupter != 0 && this->status.interruptedBy.name[0] == 0) {
				if(this->setup.status.interruptedBy) brdkStrCpy((unsigned long)this->status.interruptedBy.name,(unsigned long)((brdkEM_typ*)this->internal.pInterrupter)->status.name);
				if(this->internal.pInterrupter != (unsigned long)this) {
					this->status.interruptedBy.state = ((brdkEM_typ*)this->internal.pInterrupter)->status.interruptedBy.state;
					this->status.interruptedBy.substate = ((brdkEM_typ*)this->internal.pInterrupter)->status.interruptedBy.substate;
				}
				else {
					this->status.interruptedBy.state = ((brdkEM_typ*)this->internal.pInterrupter)->internal.old.state;
					this->status.interruptedBy.substate = ((brdkEM_typ*)this->internal.pInterrupter)->internal.old.substate;
				}
				if(this->state == STATE_ABORTING || this->state == STATE_STOPPING) {
					if(this->setup.status.last) {
						brdkStrMemMove((unsigned long)this->status.last[1],(unsigned long)this->status.last[0], sizeof(this->status.last[0])*BRDK_MU_MAX_LAST_SIZE);
						if(this->state == STATE_ABORTING) brdkStrCpy((unsigned long)this->status.last[0],(unsigned long)"Aborted by: ");
						else brdkStrCpy((unsigned long)this->status.last[0],(unsigned long)"Stopped by: ");
						brdkStrCat((unsigned long)this->status.last[0],(unsigned long)this->status.interruptedBy.name);
						brdkStrCat((unsigned long)this->status.last[0],(unsigned long)": ");
						brdkStrCat((unsigned long)this->status.last[0],brdkEMStateToA(this->status.interruptedBy.state));
						brdkStrCat((unsigned long)this->status.last[0],(unsigned long)": ");
						brdkStrAppendUdintToA(this->status.interruptedBy.substate,(unsigned long)this->status.last[0],BRDK_STR_CONVERT_DECIMAL,-1);
					}
				}
			}
			this->internal.cmdSC = this->cmd.sc = this->cmd.start = this->cmd.reset = this->cmd.abort = this->cmd.stop = this->cmd.clear = this->cmd.hold = this->cmd.complete = this->cmd.suspend = false; /* reset commands when the state changes */
			this->substate = 0;	/* reset substate by a state change */
			this->status.time = 0;
			this->status.unvalidatedMode = false;
		}
		this->status.substate[0] = this->description[0] = 0;		/* reset sub state text and description */
		this->internal.old.state = this->state;
		this->internal.old.substate = this->substate;

	}

	/* update parent info */
	if(parent != NULL) {
		this->status.parent.state = parent->state;
		this->status.parent.substate = parent->substate;
		this->status.parent.sleeping = parent->status.sleeping;
		this->status.parent.mode = parent->mode;
		this->status.parent.sc = parent->cmd.sc;
		if(parent->setup.skipStopSC) this->setup.skipStopSC = true; /* check if skipStopSC is set in parent module */
	}

	/* reactTo has changed */
	if(this->internal.old.reactTo != this->setup.reactTo) {
		if(this->setup.reactTo == BRDK_EM_REACT_TO_ALL) {
			if(parent != NULL) this->internal.findParent = true;
		}
		this->internal.old.reactTo = this->setup.reactTo;
	}

	/* update siblings info */
	updateSiblingInfo(&this->internal.muList.siblingIdx, &this->status.sibling[0]);

	/* save the restore information */
	if(this->setup.restore.activate) {
		if(this->setup.restore.pRestoreStruct != 0) {
			this->setup.restore.pRestoreStruct->mode = this->mode;
			this->setup.restore.pRestoreStruct->state = this->state;
			this->setup.restore.pRestoreStruct->substate = this->substate;
			this->setup.restore.pRestoreStruct->sc = this->internal.cmdSC;
		}
	}
}
```
